(* Schneider Machine Expert - Basic project AWGC_ALGORITMA_COMMISSIONING, file version 3.0.0.0 *)
(* ProjectInformations: Name=New project *)

HARDWARE
  Cpu 0: TM221CE24R
  ModuleExtensionObject 0: TM3DI32K
  ModuleExtensionObject 1: TM3AI2H/G
  EthernetConfiguration: NetworkName=M221, IpAllocationMode=FixedAddress, IpAddress=0.0.0.0, SubnetMask=0.0.0.0
  SerialLineConfiguration: Baud=Baud19200, Parity=ParityEven, DataBits=DataBits8, StopBits=StopBits1, PhysicalMedium=PhysicalMediumRs485, TransmissionMode=TransmissionModeModbusRtu, SlaveId=1, Addressing=SlaveAddressing
  MastTask: UsePeriodScanMode=false, PeriodScan=100
  FastTask: Period=255
  CpuBehavior: StartingMode=StartAsPreviousState, AutoSaveRamOnEeprom=true, WatchdogPeriod=250

SYMBOLS  (address, symbol, comment, settings)
  %M0       SYSTEM_ENABLE  "Izin umum gerak"
  %M1       WATER_FAULT  "Fault sinyal level"
  %M2       FAULT_G1  "Fault pintu 1"
  %M3       FAULT_G2  "Fault pintu 2"
  %M4       FAULT_G3  "Fault pintu 3"
  %M5       SCADA_COMMISSIONING_OK  "Tombol SCADA commissioning OK"
  %M10      REVERSE_G1  "Arah encoder pintu 1 dibalik"
  %M11      REVERSE_G2  "Arah encoder pintu 2 dibalik"
  %M12      REVERSE_G3  "Arah encoder pintu 3 dibalik"
  %M100     G1_BIN_B0  "Binary bit 0 hasil Gray pintu 1"
  %M101     G1_BIN_B1  "Binary bit 1 hasil Gray pintu 1"
  %M102     G1_BIN_B2  "Binary bit 2 hasil Gray pintu 1"
  %M103     G1_BIN_B3  "Binary bit 3 hasil Gray pintu 1"
  %M104     G1_BIN_B4  "Binary bit 4 hasil Gray pintu 1"
  %M105     G1_BIN_B5  "Binary bit 5 hasil Gray pintu 1"
  %M106     G1_BIN_B6  "Binary bit 6 hasil Gray pintu 1"
  %M107     G1_BIN_B7  "Binary bit 7 hasil Gray pintu 1"
  %M110     G2_BIN_B0  "Binary bit 0 hasil Gray pintu 2"
  %M111     G2_BIN_B1  "Binary bit 1 hasil Gray pintu 2"
  %M112     G2_BIN_B2  "Binary bit 2 hasil Gray pintu 2"
  %M113     G2_BIN_B3  "Binary bit 3 hasil Gray pintu 2"
  %M114     G2_BIN_B4  "Binary bit 4 hasil Gray pintu 2"
  %M115     G2_BIN_B5  "Binary bit 5 hasil Gray pintu 2"
  %M116     G2_BIN_B6  "Binary bit 6 hasil Gray pintu 2"
  %M117     G2_BIN_B7  "Binary bit 7 hasil Gray pintu 2"
  %M120     G3_BIN_B0  "Binary bit 0 hasil Gray pintu 3"
  %M121     G3_BIN_B1  "Binary bit 1 hasil Gray pintu 3"
  %M122     G3_BIN_B2  "Binary bit 2 hasil Gray pintu 3"
  %M123     G3_BIN_B3  "Binary bit 3 hasil Gray pintu 3"
  %M124     G3_BIN_B4  "Binary bit 4 hasil Gray pintu 3"
  %M125     G3_BIN_B5  "Binary bit 5 hasil Gray pintu 3"
  %M126     G3_BIN_B6  "Binary bit 6 hasil Gray pintu 3"
  %M127     G3_BIN_B7  "Binary bit 7 hasil Gray pintu 3"
  %M200     AUTO_OPEN_REQ_G1  "Request auto buka G1"
  %M201     AUTO_CLOSE_REQ_G1  "Request auto tutup G1"
  %M202     AUTO_OPEN_REQ_G2  "Request auto buka G2"
  %M203     AUTO_CLOSE_REQ_G2  "Request auto tutup G2"
  %M204     AUTO_OPEN_REQ_G3  "Request auto buka G3"
  %M205     AUTO_CLOSE_REQ_G3  "Request auto tutup G3"
  %M210     MAN_OPEN_REQ_G1  "Request manual buka G1"
  %M211     MAN_CLOSE_REQ_G1  "Request manual tutup G1"
  %M212     MAN_OPEN_REQ_G2  "Request manual buka G2"
  %M213     MAN_CLOSE_REQ_G2  "Request manual tutup G2"
  %M214     MAN_OPEN_REQ_G3  "Request manual buka G3"
  %M215     MAN_CLOSE_REQ_G3  "Request manual tutup G3"
  %M6       SCADA_STOP  "BOOL RW: 1=STOP, 0=release stop; reset to STOP on first RUN"
  %M300     SCADA_SAFETY_OK  "Virtual input Safety OK dari SCADA"
  %M301     SCADA_LS_CLOSE_G1  "Virtual limit close gate 1"
  %M302     SCADA_LS_OPEN_G1  "Virtual limit open gate 1"
  %M303     SCADA_LS_CLOSE_G2  "Virtual limit close gate 2"
  %M304     SCADA_LS_OPEN_G2  "Virtual limit open gate 2"
  %M305     SCADA_LS_CLOSE_G3  "Virtual limit close gate 3"
  %M306     SCADA_LS_OPEN_G3  "Virtual limit open gate 3"
  %M307     SCADA_OL_G1_OK  "Virtual overload gate 1 OK"
  %M308     SCADA_OL_G2_OK  "Virtual overload gate 2 OK"
  %M309     SCADA_OL_G3_OK  "Virtual overload gate 3 OK"
  %M310     SIM_I0_10  "SIM ONLY virtual physical input I0.10"
  %M311     SIM_I0_11  "SIM ONLY virtual physical input I0.11"
  %M312     SIM_I0_12  "SIM ONLY virtual physical input I0.12"
  %M313     SIM_I0_13  "SIM ONLY virtual physical input I0.13"
  %M344     SCADA_MODE_AUTO  "Virtual mode AUTO dari SCADA"
  %M345     SIM_I1_25  "SIM ONLY virtual physical input I1.25"
  %M346     SIM_I1_26  "SIM ONLY virtual physical input I1.26"
  %M347     SIM_I1_27  "SIM ONLY virtual physical input I1.27"
  %M348     SIM_I1_28  "SIM ONLY virtual physical input I1.28"
  %M349     SIM_I1_29  "SIM ONLY virtual physical input I1.29"
  %M350     SIM_I1_30  "SIM ONLY virtual physical input I1.30"
  %M351     SCADA_RESET_FAULT  "Virtual reset fault dari SCADA"
  %M360     SIM_Q0_0  "SIM ONLY output mirror Q0.0; actual output always OFF"
  %M361     SIM_Q0_1  "SIM ONLY output mirror Q0.1; actual output always OFF"
  %M362     SIM_Q0_2  "SIM ONLY output mirror Q0.2; actual output always OFF"
  %M363     SIM_Q0_3  "SIM ONLY output mirror Q0.3; actual output always OFF"
  %M364     SIM_Q0_4  "SIM ONLY output mirror Q0.4; actual output always OFF"
  %M365     SIM_Q0_5  "SIM ONLY output mirror Q0.5; actual output always OFF"
  %M320     SIM_I1_0  "SIM ONLY virtual physical input I1.0"
  %M321     SIM_I1_1  "SIM ONLY virtual physical input I1.1"
  %M322     SIM_I1_2  "SIM ONLY virtual physical input I1.2"
  %M323     SIM_I1_3  "SIM ONLY virtual physical input I1.3"
  %M324     SIM_I1_4  "SIM ONLY virtual physical input I1.4"
  %M325     SIM_I1_5  "SIM ONLY virtual physical input I1.5"
  %M326     SIM_I1_6  "SIM ONLY virtual physical input I1.6"
  %M327     SIM_I1_7  "SIM ONLY virtual physical input I1.7"
  %M328     SIM_I1_8  "SIM ONLY virtual physical input I1.8"
  %M329     SIM_I1_9  "SIM ONLY virtual physical input I1.9"
  %M330     SIM_I1_10  "SIM ONLY virtual physical input I1.10"
  %M331     SIM_I1_11  "SIM ONLY virtual physical input I1.11"
  %M332     SIM_I1_12  "SIM ONLY virtual physical input I1.12"
  %M333     SIM_I1_13  "SIM ONLY virtual physical input I1.13"
  %M334     SIM_I1_14  "SIM ONLY virtual physical input I1.14"
  %M335     SIM_I1_15  "SIM ONLY virtual physical input I1.15"
  %M336     SIM_I1_16  "SIM ONLY virtual physical input I1.16"
  %M337     SIM_I1_17  "SIM ONLY virtual physical input I1.17"
  %M338     SIM_I1_18  "SIM ONLY virtual physical input I1.18"
  %M339     SIM_I1_19  "SIM ONLY virtual physical input I1.19"
  %M340     SIM_I1_20  "SIM ONLY virtual physical input I1.20"
  %M341     SIM_I1_21  "SIM ONLY virtual physical input I1.21"
  %M342     SIM_I1_22  "SIM ONLY virtual physical input I1.22"
  %M343     SIM_I1_23  "SIM ONLY virtual physical input I1.23"
  %M366     SIM_Q0_6  "SIM ONLY output mirror Q0.6; actual output always OFF"
  %M367     SIM_Q0_7  "SIM ONLY output mirror Q0.7; actual output always OFF"
  %M368     SIM_Q0_8  "SIM ONLY output mirror Q0.8; actual output always OFF"
  %M369     SIM_Q0_9  "SIM ONLY output mirror Q0.9; actual output always OFF"
  %M370     SCADA_ENABLE_SIM  "Virtual enable simulator dari SCADA"
  %S13      SB_FIRSTRUN  "Indicates the first controller cycle in RUN mode"
  %MW1      WATER_RANGE_MM  "Range sensor level mm"
  %MW2      LEVEL_RAW_COPY  "Salinan raw input level"
  %MW10     MAX_HEIGHT_G1_MM  "Tinggi maksimum pintu 1 mm"
  %MW11     MAX_HEIGHT_G2_MM  "Tinggi maksimum pintu 2 mm"
  %MW12     MAX_HEIGHT_G3_MM  "Tinggi maksimum pintu 3 mm"
  %MW13     DEADBAND_PCT  "Deadband posisi persen"
  %MW20     ENC_ZERO_G1  "Nilai encoder pintu 1 saat tertutup"
  %MW21     ENC_ZERO_G2  "Nilai encoder pintu 2 saat tertutup"
  %MW22     ENC_ZERO_G3  "Nilai encoder pintu 3 saat tertutup"
  %MW23     ENC_SPAN_G1  "Span count tertutup-terbuka G1"
  %MW24     ENC_SPAN_G2  "Span count tertutup-terbuka G2"
  %MW25     ENC_SPAN_G3  "Span count tertutup-terbuka G3"
  %MW30     ENC_BINARY_G1  "Nilai biner encoder G1"
  %MW31     ENC_BINARY_G2  "Nilai biner encoder G2"
  %MW32     ENC_BINARY_G3  "Nilai biner encoder G3"
  %MW33     POS_COUNT_G1  "Count posisi terkoreksi G1"
  %MW34     POS_COUNT_G2  "Count posisi terkoreksi G2"
  %MW35     POS_COUNT_G3  "Count posisi terkoreksi G3"
  %MW50     TARGET_PCT_G1  "Target bukaan G1 0-100 persen"
  %MW51     TARGET_PCT_G2  "Target bukaan G2 0-100 persen"
  %MW52     TARGET_PCT_G3  "Target bukaan G3 0-100 persen"
  %MW110    SIM_PROFILE_ID  "221 identifies simulation-only project"
  %MW111    SIM_PROFILE_VERSION  "4001 identifies simulation input mapping"
  %MF60     POSITION_G1_PCT  "Posisi G1 persen"
  %MF62     POSITION_G2_PCT  "Posisi G2 persen"
  %MF64     POSITION_G3_PCT  "Posisi G3 persen"
  %MF66     POSITION_G1_MM  "Posisi G1 mm"
  %MF68     POSITION_G2_MM  "Posisi G2 mm"
  %MF70     POSITION_G3_MM  "Posisi G3 mm"
  %MF72     WATER_LEVEL_MM  "Level air mm"
  %MF74     WATER_LEVEL_PCT  "Level air persen"
  %MF76     WATER_RANGE_REAL  "Range level dalam REAL"
  %MF80     TARGET_G1_REAL  "Target G1 dalam REAL"
  %MF82     TARGET_G2_REAL  "Target G2 dalam REAL"
  %MF84     TARGET_G3_REAL  "Target G3 dalam REAL"
  %MF86     DEADBAND_REAL  "Deadband dalam REAL"
  %MF88     OPEN_THRESHOLD_G1  "Ambang buka G1"
  %MF90     CLOSE_THRESHOLD_G1  "Ambang tutup G1"
  %MF92     OPEN_THRESHOLD_G2  "Ambang buka G2"
  %MF94     CLOSE_THRESHOLD_G2  "Ambang tutup G2"
  %MF96     OPEN_THRESHOLD_G3  "Ambang buka G3"
  %MF98     CLOSE_THRESHOLD_G3  "Ambang tutup G3"
  %I0.0     SAFETY_OK_IN  "Feedback rangkaian safety hardwired sehat"
  %I0.1     LS_CLOSE_G1  "Limit tertutup pintu 1"
  %I0.2     LS_OPEN_G1  "Limit terbuka pintu 1"
  %I0.3     LS_CLOSE_G2  "Limit tertutup pintu 2"
  %I0.4     LS_OPEN_G2  "Limit terbuka pintu 2"
  %I0.5     LS_CLOSE_G3  "Limit tertutup pintu 3"
  %I0.6     LS_OPEN_G3  "Limit terbuka pintu 3"
  %I0.7     OL_OK_G1  "Overload motor pintu 1 sehat"
  %I0.8     OL_OK_G2  "Overload motor pintu 2 sehat"
  %I0.9     OL_OK_G3  "Overload motor pintu 3 sehat"
  %I0.10    SPARE_I010  "Cadangan input"
  %I0.11    SPARE_I011  "Cadangan input"
  %I0.12    SPARE_I012  "Cadangan input"
  %I0.13    SPARE_I013  "Cadangan input"
  %Q0.0     OPEN_G1  "Relay kontaktor OPEN pintu 1"
  %Q0.1     CLOSE_G1  "Relay kontaktor CLOSE pintu 1"
  %Q0.2     OPEN_G2  "Relay kontaktor OPEN pintu 2"
  %Q0.3     CLOSE_G2  "Relay kontaktor CLOSE pintu 2"
  %Q0.4     OPEN_G3  "Relay kontaktor OPEN pintu 3"
  %Q0.5     CLOSE_G3  "Relay kontaktor CLOSE pintu 3"
  %I1.0     ENC_G1_GRAY_B0  "E6CP pintu 1 Gray bit 0"
  %I1.1     ENC_G1_GRAY_B1  "E6CP pintu 1 Gray bit 1"
  %I1.2     ENC_G1_GRAY_B2  "E6CP pintu 1 Gray bit 2"
  %I1.3     ENC_G1_GRAY_B3  "E6CP pintu 1 Gray bit 3"
  %I1.4     ENC_G1_GRAY_B4  "E6CP pintu 1 Gray bit 4"
  %I1.5     ENC_G1_GRAY_B5  "E6CP pintu 1 Gray bit 5"
  %I1.6     ENC_G1_GRAY_B6  "E6CP pintu 1 Gray bit 6"
  %I1.7     ENC_G1_GRAY_B7  "E6CP pintu 1 Gray bit 7"
  %I1.8     ENC_G2_GRAY_B0  "E6CP pintu 2 Gray bit 0"
  %I1.9     ENC_G2_GRAY_B1  "E6CP pintu 2 Gray bit 1"
  %I1.10    ENC_G2_GRAY_B2  "E6CP pintu 2 Gray bit 2"
  %I1.11    ENC_G2_GRAY_B3  "E6CP pintu 2 Gray bit 3"
  %I1.12    ENC_G2_GRAY_B4  "E6CP pintu 2 Gray bit 4"
  %I1.13    ENC_G2_GRAY_B5  "E6CP pintu 2 Gray bit 5"
  %I1.14    ENC_G2_GRAY_B6  "E6CP pintu 2 Gray bit 6"
  %I1.15    ENC_G2_GRAY_B7  "E6CP pintu 2 Gray bit 7"
  %I1.16    ENC_G3_GRAY_B0  "E6CP pintu 3 Gray bit 0"
  %I1.17    ENC_G3_GRAY_B1  "E6CP pintu 3 Gray bit 1"
  %I1.18    ENC_G3_GRAY_B2  "E6CP pintu 3 Gray bit 2"
  %I1.19    ENC_G3_GRAY_B3  "E6CP pintu 3 Gray bit 3"
  %I1.20    ENC_G3_GRAY_B4  "E6CP pintu 3 Gray bit 4"
  %I1.21    ENC_G3_GRAY_B5  "E6CP pintu 3 Gray bit 5"
  %I1.22    ENC_G3_GRAY_B6  "E6CP pintu 3 Gray bit 6"
  %I1.23    ENC_G3_GRAY_B7  "E6CP pintu 3 Gray bit 7"
  %I1.24    MODE_AUTO  "Selector 1=AUTO 0=MANUAL"
  %I1.25    MAN_OPEN_G1  "PB manual buka pintu 1"
  %I1.26    MAN_CLOSE_G1  "PB manual tutup pintu 1"
  %I1.27    MAN_OPEN_G2  "PB manual buka pintu 2"
  %I1.28    MAN_CLOSE_G2  "PB manual tutup pintu 2"
  %I1.29    MAN_OPEN_G3  "PB manual buka pintu 3"
  %I1.30    MAN_CLOSE_G3  "PB manual tutup pintu 3"
  %I1.31    RESET_FAULT  "PB reset fault"
  %IW2.0    LEVEL_RAW  "Sensor level 4-20 mA raw 4000-20000"  [Type=Type_4_20mA, Scope=Scope_Customized, Minimum=4000, Maximum=20000]

POU AWGC_3_PINTU_IL
  (* SectionNumber=1 *)

// Rung 0: SIM_COLD_RESET_M369
// SIMULATOR ONLY. Physical outputs forced OFF. Do not use for plant operation.
  LD %S13                 (* SB_FIRSTRUN *)
  R %M369                 (* SIM_Q0_9 *)
  // as ST:
  //   IF SB_FIRSTRUN THEN SIM_Q0_9 := FALSE; END_IF;

// Rung 1: SIM_COLD_RESET_M368
// SIMULATOR ONLY. Physical outputs forced OFF. Do not use for plant operation.
  LD %S13                 (* SB_FIRSTRUN *)
  R %M368                 (* SIM_Q0_8 *)
  // as ST:
  //   IF SB_FIRSTRUN THEN SIM_Q0_8 := FALSE; END_IF;

// Rung 2: SIM_COLD_RESET_M367
// SIMULATOR ONLY. Physical outputs forced OFF. Do not use for plant operation.
  LD %S13                 (* SB_FIRSTRUN *)
  R %M367                 (* SIM_Q0_7 *)
  // as ST:
  //   IF SB_FIRSTRUN THEN SIM_Q0_7 := FALSE; END_IF;

// Rung 3: SIM_COLD_RESET_M366
// SIMULATOR ONLY. Physical outputs forced OFF. Do not use for plant operation.
  LD %S13                 (* SB_FIRSTRUN *)
  R %M366                 (* SIM_Q0_6 *)
  // as ST:
  //   IF SB_FIRSTRUN THEN SIM_Q0_6 := FALSE; END_IF;

// Rung 4: SIM_COLD_RESET_M365
// SIMULATOR ONLY. Physical outputs forced OFF. Do not use for plant operation.
  LD %S13                 (* SB_FIRSTRUN *)
  R %M365                 (* SIM_Q0_5 *)
  // as ST:
  //   IF SB_FIRSTRUN THEN SIM_Q0_5 := FALSE; END_IF;

// Rung 5: SIM_COLD_RESET_M364
// SIMULATOR ONLY. Physical outputs forced OFF. Do not use for plant operation.
  LD %S13                 (* SB_FIRSTRUN *)
  R %M364                 (* SIM_Q0_4 *)
  // as ST:
  //   IF SB_FIRSTRUN THEN SIM_Q0_4 := FALSE; END_IF;

// Rung 6: SIM_COLD_RESET_M363
// SIMULATOR ONLY. Physical outputs forced OFF. Do not use for plant operation.
  LD %S13                 (* SB_FIRSTRUN *)
  R %M363                 (* SIM_Q0_3 *)
  // as ST:
  //   IF SB_FIRSTRUN THEN SIM_Q0_3 := FALSE; END_IF;

// Rung 7: SIM_COLD_RESET_M362
// SIMULATOR ONLY. Physical outputs forced OFF. Do not use for plant operation.
  LD %S13                 (* SB_FIRSTRUN *)
  R %M362                 (* SIM_Q0_2 *)
  // as ST:
  //   IF SB_FIRSTRUN THEN SIM_Q0_2 := FALSE; END_IF;

// Rung 8: SIM_COLD_RESET_M361
// SIMULATOR ONLY. Physical outputs forced OFF. Do not use for plant operation.
  LD %S13                 (* SB_FIRSTRUN *)
  R %M361                 (* SIM_Q0_1 *)
  // as ST:
  //   IF SB_FIRSTRUN THEN SIM_Q0_1 := FALSE; END_IF;

// Rung 9: SIM_COLD_RESET_M360
// SIMULATOR ONLY. Physical outputs forced OFF. Do not use for plant operation.
  LD %S13                 (* SB_FIRSTRUN *)
  R %M360                 (* SIM_Q0_0 *)
  // as ST:
  //   IF SB_FIRSTRUN THEN SIM_Q0_0 := FALSE; END_IF;

// Rung 10: SIM_COLD_RESET_M351
// SIMULATOR ONLY. Physical outputs forced OFF. Do not use for plant operation.
  LD %S13                 (* SB_FIRSTRUN *)
  R %M351                 (* SCADA_RESET_FAULT *)
  // as ST:
  //   IF SB_FIRSTRUN THEN SCADA_RESET_FAULT := FALSE; END_IF;

// Rung 11: SIM_COLD_RESET_M350
// SIMULATOR ONLY. Physical outputs forced OFF. Do not use for plant operation.
  LD %S13                 (* SB_FIRSTRUN *)
  R %M350                 (* SIM_I1_30 *)
  // as ST:
  //   IF SB_FIRSTRUN THEN SIM_I1_30 := FALSE; END_IF;

// Rung 12: SIM_COLD_RESET_M349
// SIMULATOR ONLY. Physical outputs forced OFF. Do not use for plant operation.
  LD %S13                 (* SB_FIRSTRUN *)
  R %M349                 (* SIM_I1_29 *)
  // as ST:
  //   IF SB_FIRSTRUN THEN SIM_I1_29 := FALSE; END_IF;

// Rung 13: SIM_COLD_RESET_M348
// SIMULATOR ONLY. Physical outputs forced OFF. Do not use for plant operation.
  LD %S13                 (* SB_FIRSTRUN *)
  R %M348                 (* SIM_I1_28 *)
  // as ST:
  //   IF SB_FIRSTRUN THEN SIM_I1_28 := FALSE; END_IF;

// Rung 14: SIM_COLD_RESET_M347
// SIMULATOR ONLY. Physical outputs forced OFF. Do not use for plant operation.
  LD %S13                 (* SB_FIRSTRUN *)
  R %M347                 (* SIM_I1_27 *)
  // as ST:
  //   IF SB_FIRSTRUN THEN SIM_I1_27 := FALSE; END_IF;

// Rung 15: SIM_COLD_RESET_M346
// SIMULATOR ONLY. Physical outputs forced OFF. Do not use for plant operation.
  LD %S13                 (* SB_FIRSTRUN *)
  R %M346                 (* SIM_I1_26 *)
  // as ST:
  //   IF SB_FIRSTRUN THEN SIM_I1_26 := FALSE; END_IF;

// Rung 16: SIM_COLD_RESET_M345
// SIMULATOR ONLY. Physical outputs forced OFF. Do not use for plant operation.
  LD %S13                 (* SB_FIRSTRUN *)
  R %M345                 (* SIM_I1_25 *)
  // as ST:
  //   IF SB_FIRSTRUN THEN SIM_I1_25 := FALSE; END_IF;

// Rung 17: SIM_COLD_RESET_M344
// SIMULATOR ONLY. Physical outputs forced OFF. Do not use for plant operation.
  LD %S13                 (* SB_FIRSTRUN *)
  R %M344                 (* SCADA_MODE_AUTO *)
  // as ST:
  //   IF SB_FIRSTRUN THEN SCADA_MODE_AUTO := FALSE; END_IF;

// Rung 18: SIM_COLD_RESET_M343
// SIMULATOR ONLY. Physical outputs forced OFF. Do not use for plant operation.
  LD %S13                 (* SB_FIRSTRUN *)
  R %M343                 (* SIM_I1_23 *)
  // as ST:
  //   IF SB_FIRSTRUN THEN SIM_I1_23 := FALSE; END_IF;

// Rung 19: SIM_COLD_RESET_M342
// SIMULATOR ONLY. Physical outputs forced OFF. Do not use for plant operation.
  LD %S13                 (* SB_FIRSTRUN *)
  R %M342                 (* SIM_I1_22 *)
  // as ST:
  //   IF SB_FIRSTRUN THEN SIM_I1_22 := FALSE; END_IF;

// Rung 20: SIM_COLD_RESET_M341
// SIMULATOR ONLY. Physical outputs forced OFF. Do not use for plant operation.
  LD %S13                 (* SB_FIRSTRUN *)
  R %M341                 (* SIM_I1_21 *)
  // as ST:
  //   IF SB_FIRSTRUN THEN SIM_I1_21 := FALSE; END_IF;

// Rung 21: SIM_COLD_RESET_M340
// SIMULATOR ONLY. Physical outputs forced OFF. Do not use for plant operation.
  LD %S13                 (* SB_FIRSTRUN *)
  R %M340                 (* SIM_I1_20 *)
  // as ST:
  //   IF SB_FIRSTRUN THEN SIM_I1_20 := FALSE; END_IF;

// Rung 22: SIM_COLD_RESET_M339
// SIMULATOR ONLY. Physical outputs forced OFF. Do not use for plant operation.
  LD %S13                 (* SB_FIRSTRUN *)
  R %M339                 (* SIM_I1_19 *)
  // as ST:
  //   IF SB_FIRSTRUN THEN SIM_I1_19 := FALSE; END_IF;

// Rung 23: SIM_COLD_RESET_M338
// SIMULATOR ONLY. Physical outputs forced OFF. Do not use for plant operation.
  LD %S13                 (* SB_FIRSTRUN *)
  R %M338                 (* SIM_I1_18 *)
  // as ST:
  //   IF SB_FIRSTRUN THEN SIM_I1_18 := FALSE; END_IF;

// Rung 24: SIM_COLD_RESET_M337
// SIMULATOR ONLY. Physical outputs forced OFF. Do not use for plant operation.
  LD %S13                 (* SB_FIRSTRUN *)
  R %M337                 (* SIM_I1_17 *)
  // as ST:
  //   IF SB_FIRSTRUN THEN SIM_I1_17 := FALSE; END_IF;

// Rung 25: SIM_COLD_RESET_M336
// SIMULATOR ONLY. Physical outputs forced OFF. Do not use for plant operation.
  LD %S13                 (* SB_FIRSTRUN *)
  R %M336                 (* SIM_I1_16 *)
  // as ST:
  //   IF SB_FIRSTRUN THEN SIM_I1_16 := FALSE; END_IF;

// Rung 26: SIM_COLD_RESET_M335
// SIMULATOR ONLY. Physical outputs forced OFF. Do not use for plant operation.
  LD %S13                 (* SB_FIRSTRUN *)
  R %M335                 (* SIM_I1_15 *)
  // as ST:
  //   IF SB_FIRSTRUN THEN SIM_I1_15 := FALSE; END_IF;

// Rung 27: SIM_COLD_RESET_M334
// SIMULATOR ONLY. Physical outputs forced OFF. Do not use for plant operation.
  LD %S13                 (* SB_FIRSTRUN *)
  R %M334                 (* SIM_I1_14 *)
  // as ST:
  //   IF SB_FIRSTRUN THEN SIM_I1_14 := FALSE; END_IF;

// Rung 28: SIM_COLD_RESET_M333
// SIMULATOR ONLY. Physical outputs forced OFF. Do not use for plant operation.
  LD %S13                 (* SB_FIRSTRUN *)
  R %M333                 (* SIM_I1_13 *)
  // as ST:
  //   IF SB_FIRSTRUN THEN SIM_I1_13 := FALSE; END_IF;

// Rung 29: SIM_COLD_RESET_M332
// SIMULATOR ONLY. Physical outputs forced OFF. Do not use for plant operation.
  LD %S13                 (* SB_FIRSTRUN *)
  R %M332                 (* SIM_I1_12 *)
  // as ST:
  //   IF SB_FIRSTRUN THEN SIM_I1_12 := FALSE; END_IF;

// Rung 30: SIM_COLD_RESET_M331
// SIMULATOR ONLY. Physical outputs forced OFF. Do not use for plant operation.
  LD %S13                 (* SB_FIRSTRUN *)
  R %M331                 (* SIM_I1_11 *)
  // as ST:
  //   IF SB_FIRSTRUN THEN SIM_I1_11 := FALSE; END_IF;

// Rung 31: SIM_COLD_RESET_M330
// SIMULATOR ONLY. Physical outputs forced OFF. Do not use for plant operation.
  LD %S13                 (* SB_FIRSTRUN *)
  R %M330                 (* SIM_I1_10 *)
  // as ST:
  //   IF SB_FIRSTRUN THEN SIM_I1_10 := FALSE; END_IF;

// Rung 32: SIM_COLD_RESET_M329
// SIMULATOR ONLY. Physical outputs forced OFF. Do not use for plant operation.
  LD %S13                 (* SB_FIRSTRUN *)
  R %M329                 (* SIM_I1_9 *)
  // as ST:
  //   IF SB_FIRSTRUN THEN SIM_I1_9 := FALSE; END_IF;

// Rung 33: SIM_COLD_RESET_M328
// SIMULATOR ONLY. Physical outputs forced OFF. Do not use for plant operation.
  LD %S13                 (* SB_FIRSTRUN *)
  R %M328                 (* SIM_I1_8 *)
  // as ST:
  //   IF SB_FIRSTRUN THEN SIM_I1_8 := FALSE; END_IF;

// Rung 34: SIM_COLD_RESET_M327
// SIMULATOR ONLY. Physical outputs forced OFF. Do not use for plant operation.
  LD %S13                 (* SB_FIRSTRUN *)
  R %M327                 (* SIM_I1_7 *)
  // as ST:
  //   IF SB_FIRSTRUN THEN SIM_I1_7 := FALSE; END_IF;

// Rung 35: SIM_COLD_RESET_M326
// SIMULATOR ONLY. Physical outputs forced OFF. Do not use for plant operation.
  LD %S13                 (* SB_FIRSTRUN *)
  R %M326                 (* SIM_I1_6 *)
  // as ST:
  //   IF SB_FIRSTRUN THEN SIM_I1_6 := FALSE; END_IF;

// Rung 36: SIM_COLD_RESET_M325
// SIMULATOR ONLY. Physical outputs forced OFF. Do not use for plant operation.
  LD %S13                 (* SB_FIRSTRUN *)
  R %M325                 (* SIM_I1_5 *)
  // as ST:
  //   IF SB_FIRSTRUN THEN SIM_I1_5 := FALSE; END_IF;

// Rung 37: SIM_COLD_RESET_M324
// SIMULATOR ONLY. Physical outputs forced OFF. Do not use for plant operation.
  LD %S13                 (* SB_FIRSTRUN *)
  R %M324                 (* SIM_I1_4 *)
  // as ST:
  //   IF SB_FIRSTRUN THEN SIM_I1_4 := FALSE; END_IF;

// Rung 38: SIM_COLD_RESET_M323
// SIMULATOR ONLY. Physical outputs forced OFF. Do not use for plant operation.
  LD %S13                 (* SB_FIRSTRUN *)
  R %M323                 (* SIM_I1_3 *)
  // as ST:
  //   IF SB_FIRSTRUN THEN SIM_I1_3 := FALSE; END_IF;

// Rung 39: SIM_COLD_RESET_M322
// SIMULATOR ONLY. Physical outputs forced OFF. Do not use for plant operation.
  LD %S13                 (* SB_FIRSTRUN *)
  R %M322                 (* SIM_I1_2 *)
  // as ST:
  //   IF SB_FIRSTRUN THEN SIM_I1_2 := FALSE; END_IF;

// Rung 40: SIM_COLD_RESET_M321
// SIMULATOR ONLY. Physical outputs forced OFF. Do not use for plant operation.
  LD %S13                 (* SB_FIRSTRUN *)
  R %M321                 (* SIM_I1_1 *)
  // as ST:
  //   IF SB_FIRSTRUN THEN SIM_I1_1 := FALSE; END_IF;

// Rung 41: SIM_COLD_RESET_M320
// SIMULATOR ONLY. Physical outputs forced OFF. Do not use for plant operation.
  LD %S13                 (* SB_FIRSTRUN *)
  R %M320                 (* SIM_I1_0 *)
  // as ST:
  //   IF SB_FIRSTRUN THEN SIM_I1_0 := FALSE; END_IF;

// Rung 42: SIM_COLD_RESET_M313
// SIMULATOR ONLY. Physical outputs forced OFF. Do not use for plant operation.
  LD %S13                 (* SB_FIRSTRUN *)
  R %M313                 (* SIM_I0_13 *)
  // as ST:
  //   IF SB_FIRSTRUN THEN SIM_I0_13 := FALSE; END_IF;

// Rung 43: SIM_COLD_RESET_M312
// SIMULATOR ONLY. Physical outputs forced OFF. Do not use for plant operation.
  LD %S13                 (* SB_FIRSTRUN *)
  R %M312                 (* SIM_I0_12 *)
  // as ST:
  //   IF SB_FIRSTRUN THEN SIM_I0_12 := FALSE; END_IF;

// Rung 44: SIM_COLD_RESET_M311
// SIMULATOR ONLY. Physical outputs forced OFF. Do not use for plant operation.
  LD %S13                 (* SB_FIRSTRUN *)
  R %M311                 (* SIM_I0_11 *)
  // as ST:
  //   IF SB_FIRSTRUN THEN SIM_I0_11 := FALSE; END_IF;

// Rung 45: SIM_COLD_RESET_M310
// SIMULATOR ONLY. Physical outputs forced OFF. Do not use for plant operation.
  LD %S13                 (* SB_FIRSTRUN *)
  R %M310                 (* SIM_I0_10 *)
  // as ST:
  //   IF SB_FIRSTRUN THEN SIM_I0_10 := FALSE; END_IF;

// Rung 46: SIM_COLD_RESET_M309
// SIMULATOR ONLY. Physical outputs forced OFF. Do not use for plant operation.
  LD %S13                 (* SB_FIRSTRUN *)
  R %M309                 (* SCADA_OL_G3_OK *)
  // as ST:
  //   IF SB_FIRSTRUN THEN SCADA_OL_G3_OK := FALSE; END_IF;

// Rung 47: SIM_COLD_RESET_M308
// SIMULATOR ONLY. Physical outputs forced OFF. Do not use for plant operation.
  LD %S13                 (* SB_FIRSTRUN *)
  R %M308                 (* SCADA_OL_G2_OK *)
  // as ST:
  //   IF SB_FIRSTRUN THEN SCADA_OL_G2_OK := FALSE; END_IF;

// Rung 48: SIM_COLD_RESET_M307
// SIMULATOR ONLY. Physical outputs forced OFF. Do not use for plant operation.
  LD %S13                 (* SB_FIRSTRUN *)
  R %M307                 (* SCADA_OL_G1_OK *)
  // as ST:
  //   IF SB_FIRSTRUN THEN SCADA_OL_G1_OK := FALSE; END_IF;

// Rung 49: SIM_COLD_RESET_M306
// SIMULATOR ONLY. Physical outputs forced OFF. Do not use for plant operation.
  LD %S13                 (* SB_FIRSTRUN *)
  R %M306                 (* SCADA_LS_OPEN_G3 *)
  // as ST:
  //   IF SB_FIRSTRUN THEN SCADA_LS_OPEN_G3 := FALSE; END_IF;

// Rung 50: SIM_COLD_RESET_M305
// SIMULATOR ONLY. Physical outputs forced OFF. Do not use for plant operation.
  LD %S13                 (* SB_FIRSTRUN *)
  R %M305                 (* SCADA_LS_CLOSE_G3 *)
  // as ST:
  //   IF SB_FIRSTRUN THEN SCADA_LS_CLOSE_G3 := FALSE; END_IF;

// Rung 51: SIM_COLD_RESET_M304
// SIMULATOR ONLY. Physical outputs forced OFF. Do not use for plant operation.
  LD %S13                 (* SB_FIRSTRUN *)
  R %M304                 (* SCADA_LS_OPEN_G2 *)
  // as ST:
  //   IF SB_FIRSTRUN THEN SCADA_LS_OPEN_G2 := FALSE; END_IF;

// Rung 52: SIM_COLD_RESET_M303
// SIMULATOR ONLY. Physical outputs forced OFF. Do not use for plant operation.
  LD %S13                 (* SB_FIRSTRUN *)
  R %M303                 (* SCADA_LS_CLOSE_G2 *)
  // as ST:
  //   IF SB_FIRSTRUN THEN SCADA_LS_CLOSE_G2 := FALSE; END_IF;

// Rung 53: SIM_COLD_RESET_M302
// SIMULATOR ONLY. Physical outputs forced OFF. Do not use for plant operation.
  LD %S13                 (* SB_FIRSTRUN *)
  R %M302                 (* SCADA_LS_OPEN_G1 *)
  // as ST:
  //   IF SB_FIRSTRUN THEN SCADA_LS_OPEN_G1 := FALSE; END_IF;

// Rung 54: SIM_COLD_RESET_M301
// SIMULATOR ONLY. Physical outputs forced OFF. Do not use for plant operation.
  LD %S13                 (* SB_FIRSTRUN *)
  R %M301                 (* SCADA_LS_CLOSE_G1 *)
  // as ST:
  //   IF SB_FIRSTRUN THEN SCADA_LS_CLOSE_G1 := FALSE; END_IF;

// Rung 55: SIM_COLD_RESET_M300
// SIMULATOR ONLY. Physical outputs forced OFF. Do not use for plant operation.
  LD %S13                 (* SB_FIRSTRUN *)
  R %M300                 (* SCADA_SAFETY_OK *)
  // as ST:
  //   IF SB_FIRSTRUN THEN SCADA_SAFETY_OK := FALSE; END_IF;

// Rung 56: SIM_COLD_RESET_M370
// SIMULATOR ONLY. Physical outputs forced OFF. Do not use for plant operation.
  LD %S13                 (* SB_FIRSTRUN *)
  R %M370                 (* SCADA_ENABLE_SIM *)
  // as ST:
  //   IF SB_FIRSTRUN THEN SCADA_ENABLE_SIM := FALSE; END_IF;

// Rung 57: SIM_COLD_RESET_M5
// SIMULATOR ONLY. Physical outputs forced OFF. Do not use for plant operation.
  LD %S13                 (* SB_FIRSTRUN *)
  R %M5                   (* SCADA_COMMISSIONING_OK *)
  // as ST:
  //   IF SB_FIRSTRUN THEN SCADA_COMMISSIONING_OK := FALSE; END_IF;

// Rung 58: SIM_PROFILE_ID
// SIMULATOR ONLY. Physical outputs forced OFF. Do not use for plant operation.
  LD 1
  [ %MW110 := 221 ]       (* SIM_PROFILE_ID *)
  // as ST:
  //   SIM_PROFILE_ID := 221;

// Rung 59: SIM_PROFILE_VERSION
// SIMULATOR ONLY. Physical outputs forced OFF. Do not use for plant operation.
  LD 1
  [ %MW111 := 4001 ]      (* SIM_PROFILE_VERSION *)
  // as ST:
  //   SIM_PROFILE_VERSION := 4001;

// Rung 60: REV3_SCADA_VERSION
// REV3 SCADA compatibility marker; not authentication.
  LD 1
  [ %MW111 := 3001 ]      (* SIM_PROFILE_VERSION *)
  // as ST:
  //   SIM_PROFILE_VERSION := 3001;

// Rung 61: REV3_SCADA_ID
// REV3 SCADA compatibility marker; not authentication.
  LD 1
  [ %MW110 := 221 ]       (* SIM_PROFILE_ID *)
  // as ST:
  //   SIM_PROFILE_ID := 221;

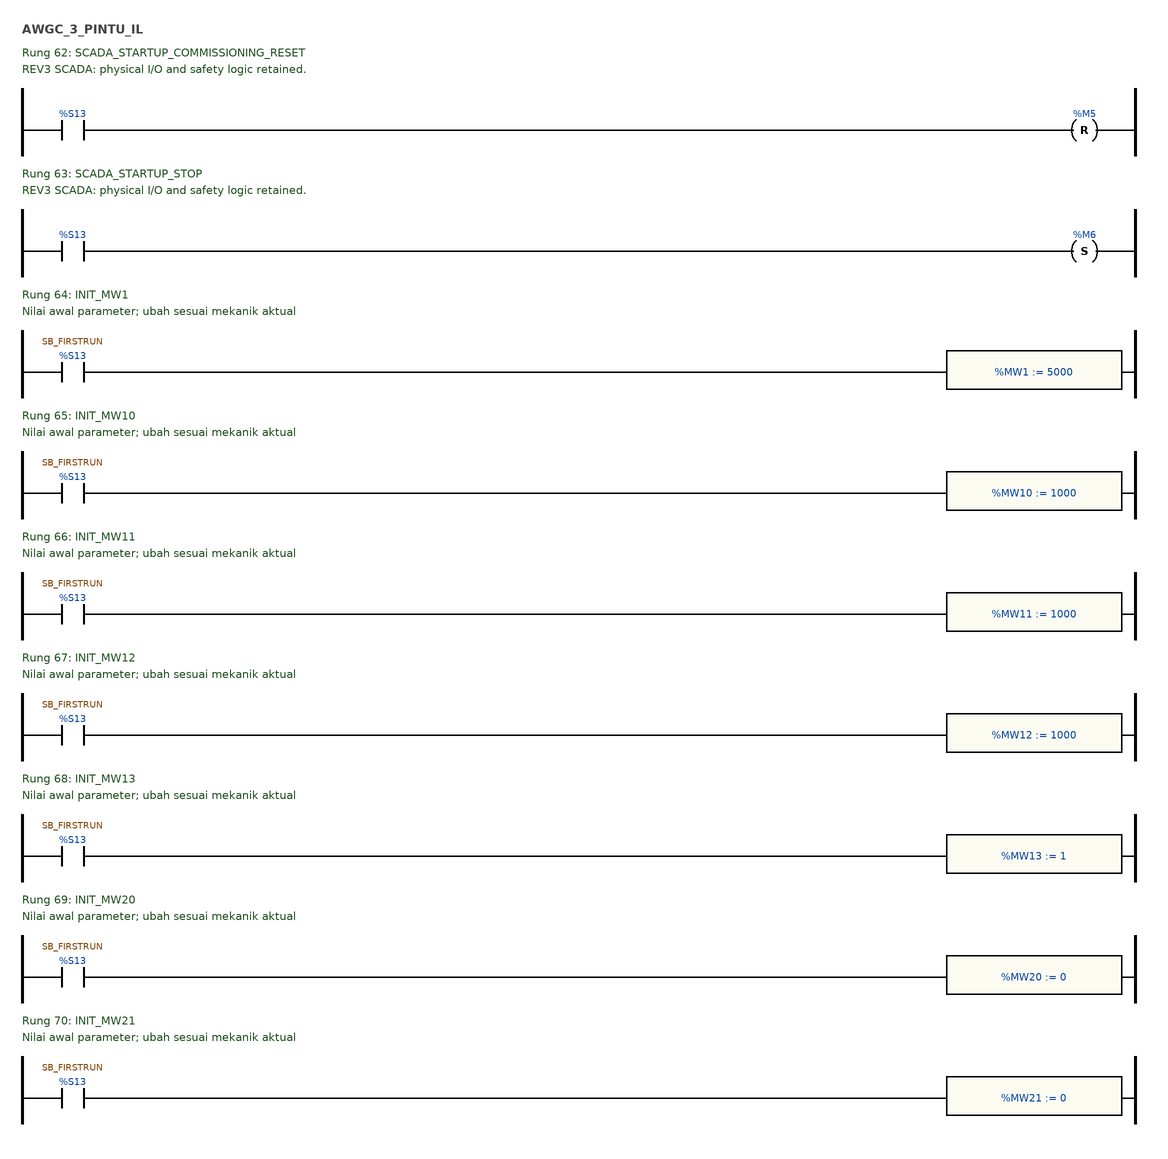

// Rung 62: SCADA_STARTUP_COMMISSIONING_RESET
// REV3 SCADA: physical I/O and safety logic retained.
  LD %S13                 (* SB_FIRSTRUN *)
  R %M5                   (* SCADA_COMMISSIONING_OK *)
  // as ST:
  //   IF SB_FIRSTRUN THEN SCADA_COMMISSIONING_OK := FALSE; END_IF;

// Rung 63: SCADA_STARTUP_STOP
// REV3 SCADA: physical I/O and safety logic retained.
  LD %S13                 (* SB_FIRSTRUN *)
  S %M6                   (* SCADA_STOP *)
  // as ST:
  //   IF SB_FIRSTRUN THEN SCADA_STOP := TRUE; END_IF;

// Rung 64: INIT_MW1
// Nilai awal parameter; ubah sesuai mekanik aktual
  LD %S13                 (* SB_FIRSTRUN *)
  [ %MW1 := 5000 ]        (* WATER_RANGE_MM *)
  // as ST:
  //   IF SB_FIRSTRUN THEN WATER_RANGE_MM := 5000; END_IF;

// Rung 65: INIT_MW10
// Nilai awal parameter; ubah sesuai mekanik aktual
  LD %S13                 (* SB_FIRSTRUN *)
  [ %MW10 := 1000 ]       (* MAX_HEIGHT_G1_MM *)
  // as ST:
  //   IF SB_FIRSTRUN THEN MAX_HEIGHT_G1_MM := 1000; END_IF;

// Rung 66: INIT_MW11
// Nilai awal parameter; ubah sesuai mekanik aktual
  LD %S13                 (* SB_FIRSTRUN *)
  [ %MW11 := 1000 ]       (* MAX_HEIGHT_G2_MM *)
  // as ST:
  //   IF SB_FIRSTRUN THEN MAX_HEIGHT_G2_MM := 1000; END_IF;

// Rung 67: INIT_MW12
// Nilai awal parameter; ubah sesuai mekanik aktual
  LD %S13                 (* SB_FIRSTRUN *)
  [ %MW12 := 1000 ]       (* MAX_HEIGHT_G3_MM *)
  // as ST:
  //   IF SB_FIRSTRUN THEN MAX_HEIGHT_G3_MM := 1000; END_IF;

// Rung 68: INIT_MW13
// Nilai awal parameter; ubah sesuai mekanik aktual
  LD %S13                 (* SB_FIRSTRUN *)
  [ %MW13 := 1 ]          (* DEADBAND_PCT *)
  // as ST:
  //   IF SB_FIRSTRUN THEN DEADBAND_PCT := 1; END_IF;

// Rung 69: INIT_MW20
// Nilai awal parameter; ubah sesuai mekanik aktual
  LD %S13                 (* SB_FIRSTRUN *)
  [ %MW20 := 0 ]          (* ENC_ZERO_G1 *)
  // as ST:
  //   IF SB_FIRSTRUN THEN ENC_ZERO_G1 := 0; END_IF;

// Rung 70: INIT_MW21
// Nilai awal parameter; ubah sesuai mekanik aktual
  LD %S13                 (* SB_FIRSTRUN *)
  [ %MW21 := 0 ]          (* ENC_ZERO_G2 *)
  // as ST:
  //   IF SB_FIRSTRUN THEN ENC_ZERO_G2 := 0; END_IF;

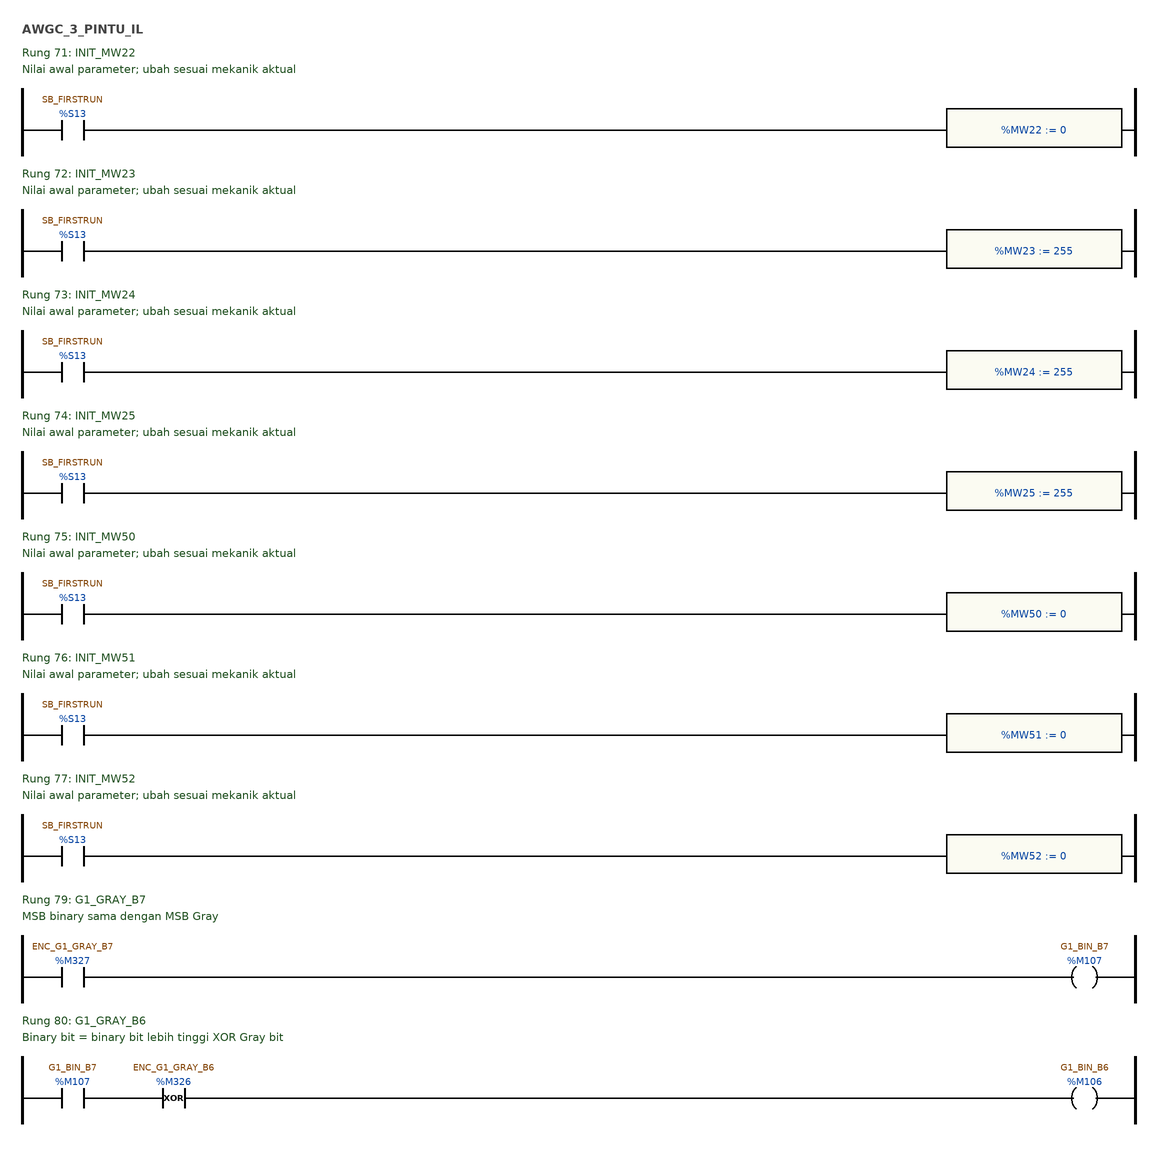

// Rung 71: INIT_MW22
// Nilai awal parameter; ubah sesuai mekanik aktual
  LD %S13                 (* SB_FIRSTRUN *)
  [ %MW22 := 0 ]          (* ENC_ZERO_G3 *)
  // as ST:
  //   IF SB_FIRSTRUN THEN ENC_ZERO_G3 := 0; END_IF;

// Rung 72: INIT_MW23
// Nilai awal parameter; ubah sesuai mekanik aktual
  LD %S13                 (* SB_FIRSTRUN *)
  [ %MW23 := 255 ]        (* ENC_SPAN_G1 *)
  // as ST:
  //   IF SB_FIRSTRUN THEN ENC_SPAN_G1 := 255; END_IF;

// Rung 73: INIT_MW24
// Nilai awal parameter; ubah sesuai mekanik aktual
  LD %S13                 (* SB_FIRSTRUN *)
  [ %MW24 := 255 ]        (* ENC_SPAN_G2 *)
  // as ST:
  //   IF SB_FIRSTRUN THEN ENC_SPAN_G2 := 255; END_IF;

// Rung 74: INIT_MW25
// Nilai awal parameter; ubah sesuai mekanik aktual
  LD %S13                 (* SB_FIRSTRUN *)
  [ %MW25 := 255 ]        (* ENC_SPAN_G3 *)
  // as ST:
  //   IF SB_FIRSTRUN THEN ENC_SPAN_G3 := 255; END_IF;

// Rung 75: INIT_MW50
// Nilai awal parameter; ubah sesuai mekanik aktual
  LD %S13                 (* SB_FIRSTRUN *)
  [ %MW50 := 0 ]          (* TARGET_PCT_G1 *)
  // as ST:
  //   IF SB_FIRSTRUN THEN TARGET_PCT_G1 := 0; END_IF;

// Rung 76: INIT_MW51
// Nilai awal parameter; ubah sesuai mekanik aktual
  LD %S13                 (* SB_FIRSTRUN *)
  [ %MW51 := 0 ]          (* TARGET_PCT_G2 *)
  // as ST:
  //   IF SB_FIRSTRUN THEN TARGET_PCT_G2 := 0; END_IF;

// Rung 77: INIT_MW52
// Nilai awal parameter; ubah sesuai mekanik aktual
  LD %S13                 (* SB_FIRSTRUN *)
  [ %MW52 := 0 ]          (* TARGET_PCT_G3 *)
  // as ST:
  //   IF SB_FIRSTRUN THEN TARGET_PCT_G3 := 0; END_IF;

// Rung 78: SYSTEM_PERMISSIVE_SIM
// SIMULATOR ONLY. Physical outputs forced OFF. Do not use for plant operation.
  LD %M300                (* SCADA_SAFETY_OK *)
  AND %M307               (* SCADA_OL_G1_OK *)
  AND %M308               (* SCADA_OL_G2_OK *)
  AND %M309               (* SCADA_OL_G3_OK *)
  AND %M5                 (* SCADA_COMMISSIONING_OK *)
  AND %M370               (* SCADA_ENABLE_SIM *)
  ST %M0                  (* SYSTEM_ENABLE *)
  // as ST:
  //   SYSTEM_ENABLE := SCADA_SAFETY_OK AND SCADA_OL_G1_OK AND SCADA_OL_G2_OK AND SCADA_OL_G3_OK AND SCADA_COMMISSIONING_OK AND SCADA_ENABLE_SIM;

// Rung 79: G1_GRAY_B7
// MSB binary sama dengan MSB Gray
  LD %M327                (* SIM_I1_7 *)
  ST %M107                (* G1_BIN_B7 *)
  // as ST:
  //   G1_BIN_B7 := SIM_I1_7;

// Rung 80: G1_GRAY_B6
// Binary bit = binary bit lebih tinggi XOR Gray bit
  LD %M107                (* G1_BIN_B7 *)
  XOR %M326               (* SIM_I1_6 *)
  ST %M106                (* G1_BIN_B6 *)
  // as ST:
  //   G1_BIN_B6 := G1_BIN_B7 XOR SIM_I1_6;

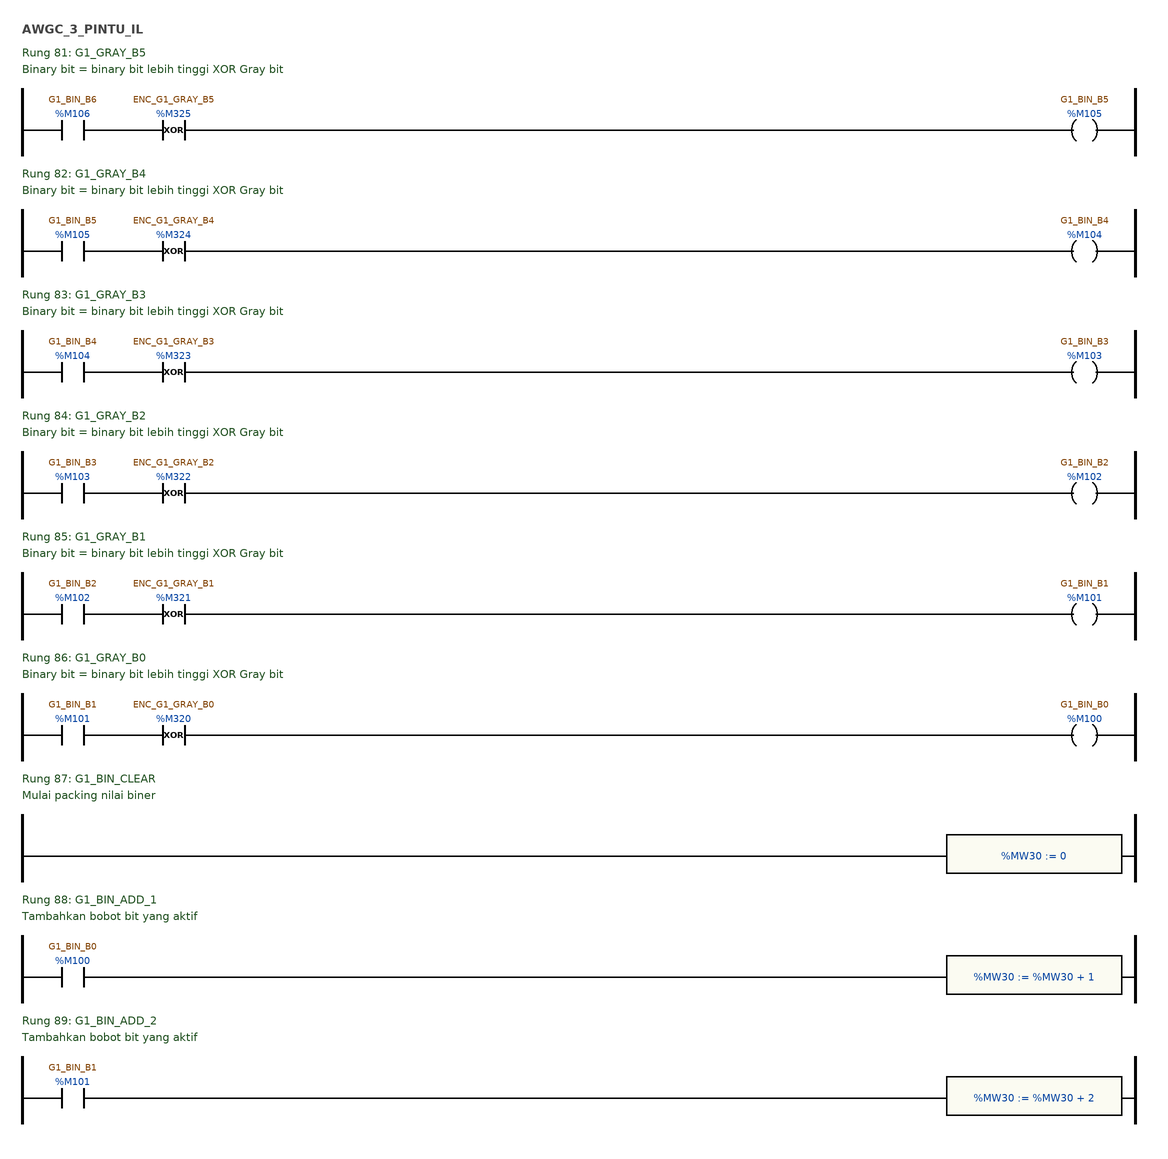

// Rung 81: G1_GRAY_B5
// Binary bit = binary bit lebih tinggi XOR Gray bit
  LD %M106                (* G1_BIN_B6 *)
  XOR %M325               (* SIM_I1_5 *)
  ST %M105                (* G1_BIN_B5 *)
  // as ST:
  //   G1_BIN_B5 := G1_BIN_B6 XOR SIM_I1_5;

// Rung 82: G1_GRAY_B4
// Binary bit = binary bit lebih tinggi XOR Gray bit
  LD %M105                (* G1_BIN_B5 *)
  XOR %M324               (* SIM_I1_4 *)
  ST %M104                (* G1_BIN_B4 *)
  // as ST:
  //   G1_BIN_B4 := G1_BIN_B5 XOR SIM_I1_4;

// Rung 83: G1_GRAY_B3
// Binary bit = binary bit lebih tinggi XOR Gray bit
  LD %M104                (* G1_BIN_B4 *)
  XOR %M323               (* SIM_I1_3 *)
  ST %M103                (* G1_BIN_B3 *)
  // as ST:
  //   G1_BIN_B3 := G1_BIN_B4 XOR SIM_I1_3;

// Rung 84: G1_GRAY_B2
// Binary bit = binary bit lebih tinggi XOR Gray bit
  LD %M103                (* G1_BIN_B3 *)
  XOR %M322               (* SIM_I1_2 *)
  ST %M102                (* G1_BIN_B2 *)
  // as ST:
  //   G1_BIN_B2 := G1_BIN_B3 XOR SIM_I1_2;

// Rung 85: G1_GRAY_B1
// Binary bit = binary bit lebih tinggi XOR Gray bit
  LD %M102                (* G1_BIN_B2 *)
  XOR %M321               (* SIM_I1_1 *)
  ST %M101                (* G1_BIN_B1 *)
  // as ST:
  //   G1_BIN_B1 := G1_BIN_B2 XOR SIM_I1_1;

// Rung 86: G1_GRAY_B0
// Binary bit = binary bit lebih tinggi XOR Gray bit
  LD %M101                (* G1_BIN_B1 *)
  XOR %M320               (* SIM_I1_0 *)
  ST %M100                (* G1_BIN_B0 *)
  // as ST:
  //   G1_BIN_B0 := G1_BIN_B1 XOR SIM_I1_0;

// Rung 87: G1_BIN_CLEAR
// Mulai packing nilai biner
  LD 1
  [ %MW30 := 0 ]          (* ENC_BINARY_G1 *)
  // as ST:
  //   ENC_BINARY_G1 := 0;

// Rung 88: G1_BIN_ADD_1
// Tambahkan bobot bit yang aktif
  LD %M100                (* G1_BIN_B0 *)
  [ %MW30 := %MW30 + 1 ]  (* ENC_BINARY_G1, ENC_BINARY_G1 *)
  // as ST:
  //   IF G1_BIN_B0 THEN ENC_BINARY_G1 := ENC_BINARY_G1 + 1; END_IF;

// Rung 89: G1_BIN_ADD_2
// Tambahkan bobot bit yang aktif
  LD %M101                (* G1_BIN_B1 *)
  [ %MW30 := %MW30 + 2 ]  (* ENC_BINARY_G1, ENC_BINARY_G1 *)
  // as ST:
  //   IF G1_BIN_B1 THEN ENC_BINARY_G1 := ENC_BINARY_G1 + 2; END_IF;

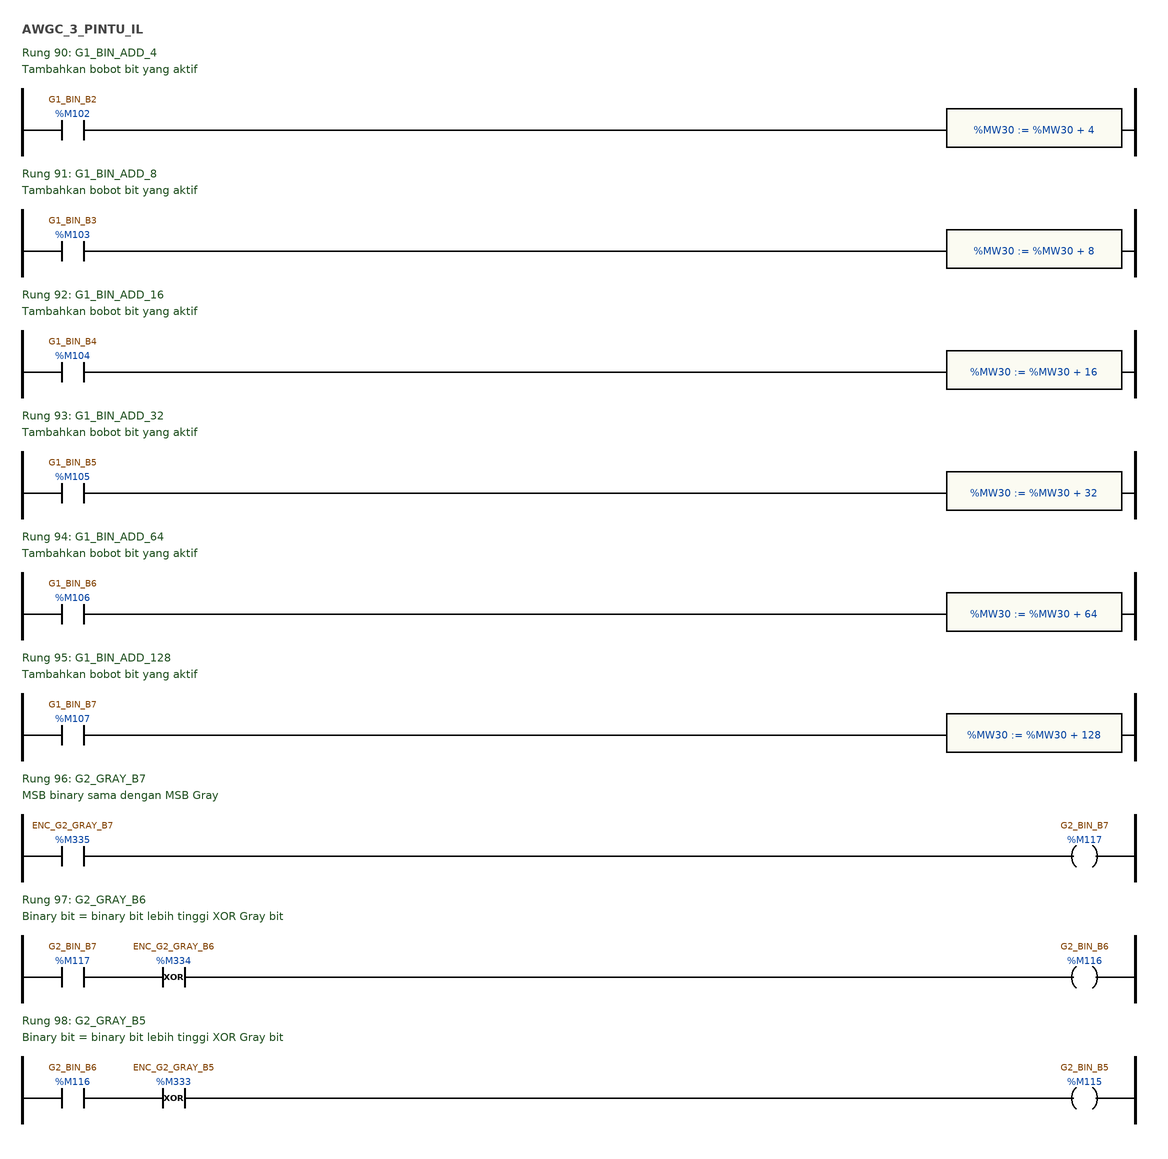

// Rung 90: G1_BIN_ADD_4
// Tambahkan bobot bit yang aktif
  LD %M102                (* G1_BIN_B2 *)
  [ %MW30 := %MW30 + 4 ]  (* ENC_BINARY_G1, ENC_BINARY_G1 *)
  // as ST:
  //   IF G1_BIN_B2 THEN ENC_BINARY_G1 := ENC_BINARY_G1 + 4; END_IF;

// Rung 91: G1_BIN_ADD_8
// Tambahkan bobot bit yang aktif
  LD %M103                (* G1_BIN_B3 *)
  [ %MW30 := %MW30 + 8 ]  (* ENC_BINARY_G1, ENC_BINARY_G1 *)
  // as ST:
  //   IF G1_BIN_B3 THEN ENC_BINARY_G1 := ENC_BINARY_G1 + 8; END_IF;

// Rung 92: G1_BIN_ADD_16
// Tambahkan bobot bit yang aktif
  LD %M104                (* G1_BIN_B4 *)
  [ %MW30 := %MW30 + 16 ] (* ENC_BINARY_G1, ENC_BINARY_G1 *)
  // as ST:
  //   IF G1_BIN_B4 THEN ENC_BINARY_G1 := ENC_BINARY_G1 + 16; END_IF;

// Rung 93: G1_BIN_ADD_32
// Tambahkan bobot bit yang aktif
  LD %M105                (* G1_BIN_B5 *)
  [ %MW30 := %MW30 + 32 ] (* ENC_BINARY_G1, ENC_BINARY_G1 *)
  // as ST:
  //   IF G1_BIN_B5 THEN ENC_BINARY_G1 := ENC_BINARY_G1 + 32; END_IF;

// Rung 94: G1_BIN_ADD_64
// Tambahkan bobot bit yang aktif
  LD %M106                (* G1_BIN_B6 *)
  [ %MW30 := %MW30 + 64 ] (* ENC_BINARY_G1, ENC_BINARY_G1 *)
  // as ST:
  //   IF G1_BIN_B6 THEN ENC_BINARY_G1 := ENC_BINARY_G1 + 64; END_IF;

// Rung 95: G1_BIN_ADD_128
// Tambahkan bobot bit yang aktif
  LD %M107                (* G1_BIN_B7 *)
  [ %MW30 := %MW30 + 128 ](* ENC_BINARY_G1, ENC_BINARY_G1 *)
  // as ST:
  //   IF G1_BIN_B7 THEN ENC_BINARY_G1 := ENC_BINARY_G1 + 128; END_IF;

// Rung 96: G2_GRAY_B7
// MSB binary sama dengan MSB Gray
  LD %M335                (* SIM_I1_15 *)
  ST %M117                (* G2_BIN_B7 *)
  // as ST:
  //   G2_BIN_B7 := SIM_I1_15;

// Rung 97: G2_GRAY_B6
// Binary bit = binary bit lebih tinggi XOR Gray bit
  LD %M117                (* G2_BIN_B7 *)
  XOR %M334               (* SIM_I1_14 *)
  ST %M116                (* G2_BIN_B6 *)
  // as ST:
  //   G2_BIN_B6 := G2_BIN_B7 XOR SIM_I1_14;

// Rung 98: G2_GRAY_B5
// Binary bit = binary bit lebih tinggi XOR Gray bit
  LD %M116                (* G2_BIN_B6 *)
  XOR %M333               (* SIM_I1_13 *)
  ST %M115                (* G2_BIN_B5 *)
  // as ST:
  //   G2_BIN_B5 := G2_BIN_B6 XOR SIM_I1_13;

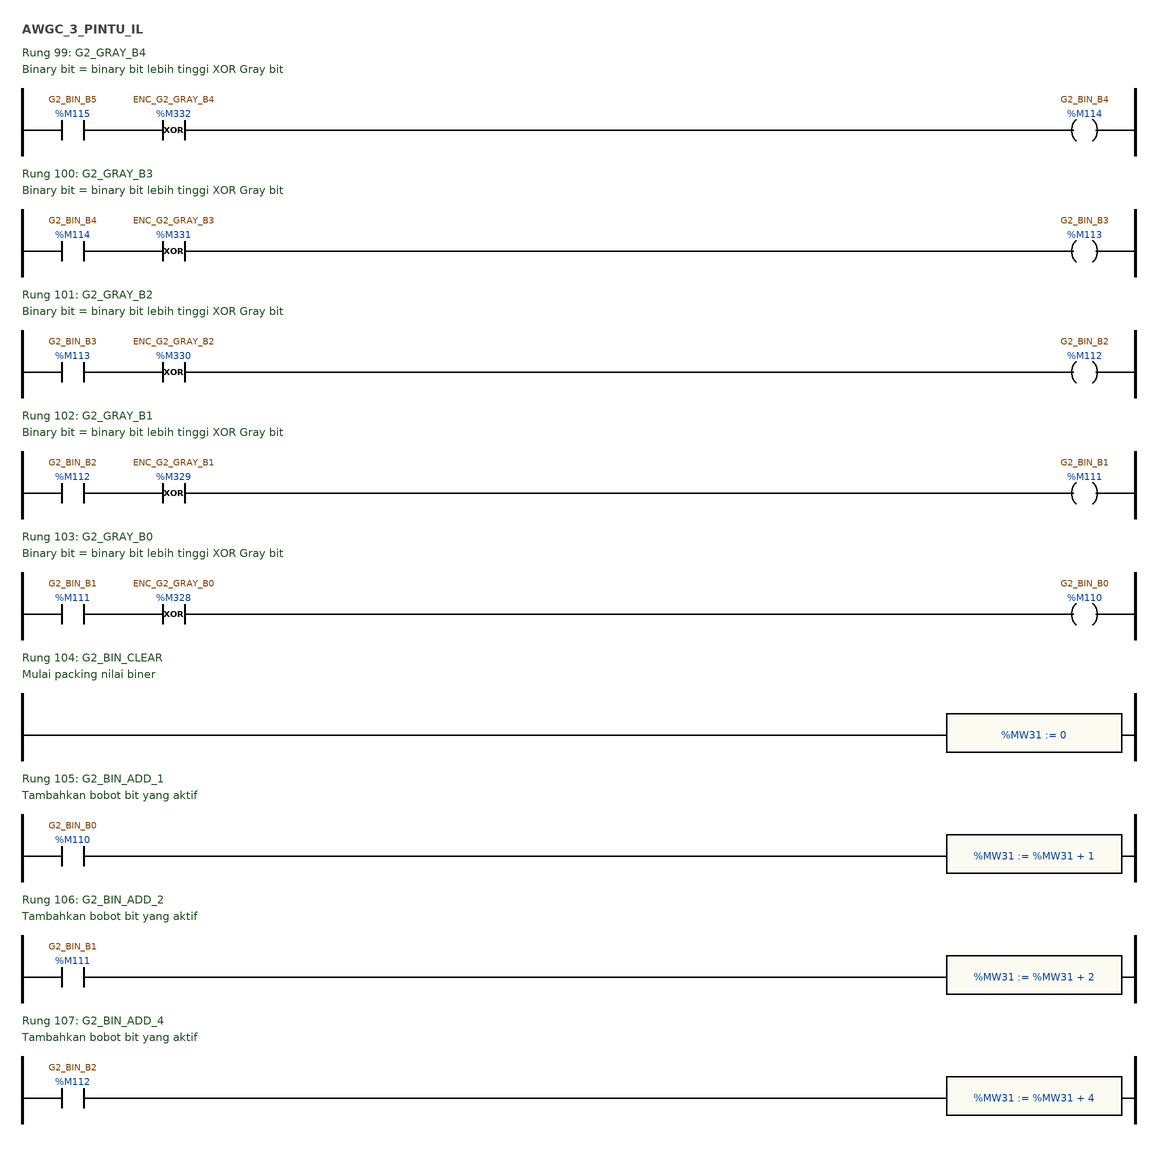

// Rung 99: G2_GRAY_B4
// Binary bit = binary bit lebih tinggi XOR Gray bit
  LD %M115                (* G2_BIN_B5 *)
  XOR %M332               (* SIM_I1_12 *)
  ST %M114                (* G2_BIN_B4 *)
  // as ST:
  //   G2_BIN_B4 := G2_BIN_B5 XOR SIM_I1_12;

// Rung 100: G2_GRAY_B3
// Binary bit = binary bit lebih tinggi XOR Gray bit
  LD %M114                (* G2_BIN_B4 *)
  XOR %M331               (* SIM_I1_11 *)
  ST %M113                (* G2_BIN_B3 *)
  // as ST:
  //   G2_BIN_B3 := G2_BIN_B4 XOR SIM_I1_11;

// Rung 101: G2_GRAY_B2
// Binary bit = binary bit lebih tinggi XOR Gray bit
  LD %M113                (* G2_BIN_B3 *)
  XOR %M330               (* SIM_I1_10 *)
  ST %M112                (* G2_BIN_B2 *)
  // as ST:
  //   G2_BIN_B2 := G2_BIN_B3 XOR SIM_I1_10;

// Rung 102: G2_GRAY_B1
// Binary bit = binary bit lebih tinggi XOR Gray bit
  LD %M112                (* G2_BIN_B2 *)
  XOR %M329               (* SIM_I1_9 *)
  ST %M111                (* G2_BIN_B1 *)
  // as ST:
  //   G2_BIN_B1 := G2_BIN_B2 XOR SIM_I1_9;

// Rung 103: G2_GRAY_B0
// Binary bit = binary bit lebih tinggi XOR Gray bit
  LD %M111                (* G2_BIN_B1 *)
  XOR %M328               (* SIM_I1_8 *)
  ST %M110                (* G2_BIN_B0 *)
  // as ST:
  //   G2_BIN_B0 := G2_BIN_B1 XOR SIM_I1_8;

// Rung 104: G2_BIN_CLEAR
// Mulai packing nilai biner
  LD 1
  [ %MW31 := 0 ]          (* ENC_BINARY_G2 *)
  // as ST:
  //   ENC_BINARY_G2 := 0;

// Rung 105: G2_BIN_ADD_1
// Tambahkan bobot bit yang aktif
  LD %M110                (* G2_BIN_B0 *)
  [ %MW31 := %MW31 + 1 ]  (* ENC_BINARY_G2, ENC_BINARY_G2 *)
  // as ST:
  //   IF G2_BIN_B0 THEN ENC_BINARY_G2 := ENC_BINARY_G2 + 1; END_IF;

// Rung 106: G2_BIN_ADD_2
// Tambahkan bobot bit yang aktif
  LD %M111                (* G2_BIN_B1 *)
  [ %MW31 := %MW31 + 2 ]  (* ENC_BINARY_G2, ENC_BINARY_G2 *)
  // as ST:
  //   IF G2_BIN_B1 THEN ENC_BINARY_G2 := ENC_BINARY_G2 + 2; END_IF;

// Rung 107: G2_BIN_ADD_4
// Tambahkan bobot bit yang aktif
  LD %M112                (* G2_BIN_B2 *)
  [ %MW31 := %MW31 + 4 ]  (* ENC_BINARY_G2, ENC_BINARY_G2 *)
  // as ST:
  //   IF G2_BIN_B2 THEN ENC_BINARY_G2 := ENC_BINARY_G2 + 4; END_IF;

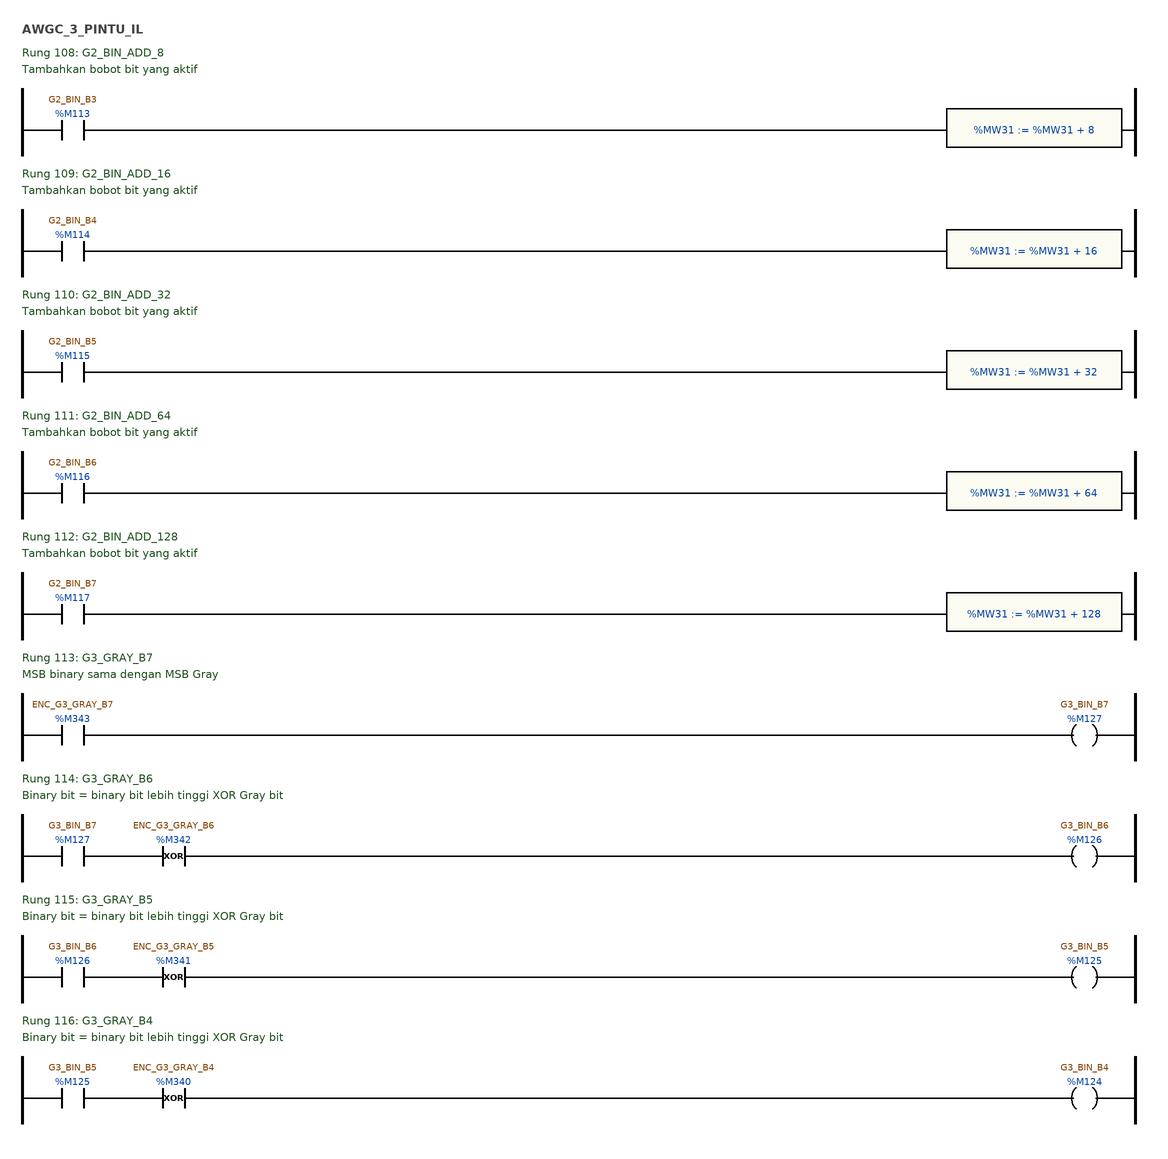

// Rung 108: G2_BIN_ADD_8
// Tambahkan bobot bit yang aktif
  LD %M113                (* G2_BIN_B3 *)
  [ %MW31 := %MW31 + 8 ]  (* ENC_BINARY_G2, ENC_BINARY_G2 *)
  // as ST:
  //   IF G2_BIN_B3 THEN ENC_BINARY_G2 := ENC_BINARY_G2 + 8; END_IF;

// Rung 109: G2_BIN_ADD_16
// Tambahkan bobot bit yang aktif
  LD %M114                (* G2_BIN_B4 *)
  [ %MW31 := %MW31 + 16 ] (* ENC_BINARY_G2, ENC_BINARY_G2 *)
  // as ST:
  //   IF G2_BIN_B4 THEN ENC_BINARY_G2 := ENC_BINARY_G2 + 16; END_IF;

// Rung 110: G2_BIN_ADD_32
// Tambahkan bobot bit yang aktif
  LD %M115                (* G2_BIN_B5 *)
  [ %MW31 := %MW31 + 32 ] (* ENC_BINARY_G2, ENC_BINARY_G2 *)
  // as ST:
  //   IF G2_BIN_B5 THEN ENC_BINARY_G2 := ENC_BINARY_G2 + 32; END_IF;

// Rung 111: G2_BIN_ADD_64
// Tambahkan bobot bit yang aktif
  LD %M116                (* G2_BIN_B6 *)
  [ %MW31 := %MW31 + 64 ] (* ENC_BINARY_G2, ENC_BINARY_G2 *)
  // as ST:
  //   IF G2_BIN_B6 THEN ENC_BINARY_G2 := ENC_BINARY_G2 + 64; END_IF;

// Rung 112: G2_BIN_ADD_128
// Tambahkan bobot bit yang aktif
  LD %M117                (* G2_BIN_B7 *)
  [ %MW31 := %MW31 + 128 ](* ENC_BINARY_G2, ENC_BINARY_G2 *)
  // as ST:
  //   IF G2_BIN_B7 THEN ENC_BINARY_G2 := ENC_BINARY_G2 + 128; END_IF;

// Rung 113: G3_GRAY_B7
// MSB binary sama dengan MSB Gray
  LD %M343                (* SIM_I1_23 *)
  ST %M127                (* G3_BIN_B7 *)
  // as ST:
  //   G3_BIN_B7 := SIM_I1_23;

// Rung 114: G3_GRAY_B6
// Binary bit = binary bit lebih tinggi XOR Gray bit
  LD %M127                (* G3_BIN_B7 *)
  XOR %M342               (* SIM_I1_22 *)
  ST %M126                (* G3_BIN_B6 *)
  // as ST:
  //   G3_BIN_B6 := G3_BIN_B7 XOR SIM_I1_22;

// Rung 115: G3_GRAY_B5
// Binary bit = binary bit lebih tinggi XOR Gray bit
  LD %M126                (* G3_BIN_B6 *)
  XOR %M341               (* SIM_I1_21 *)
  ST %M125                (* G3_BIN_B5 *)
  // as ST:
  //   G3_BIN_B5 := G3_BIN_B6 XOR SIM_I1_21;

// Rung 116: G3_GRAY_B4
// Binary bit = binary bit lebih tinggi XOR Gray bit
  LD %M125                (* G3_BIN_B5 *)
  XOR %M340               (* SIM_I1_20 *)
  ST %M124                (* G3_BIN_B4 *)
  // as ST:
  //   G3_BIN_B4 := G3_BIN_B5 XOR SIM_I1_20;

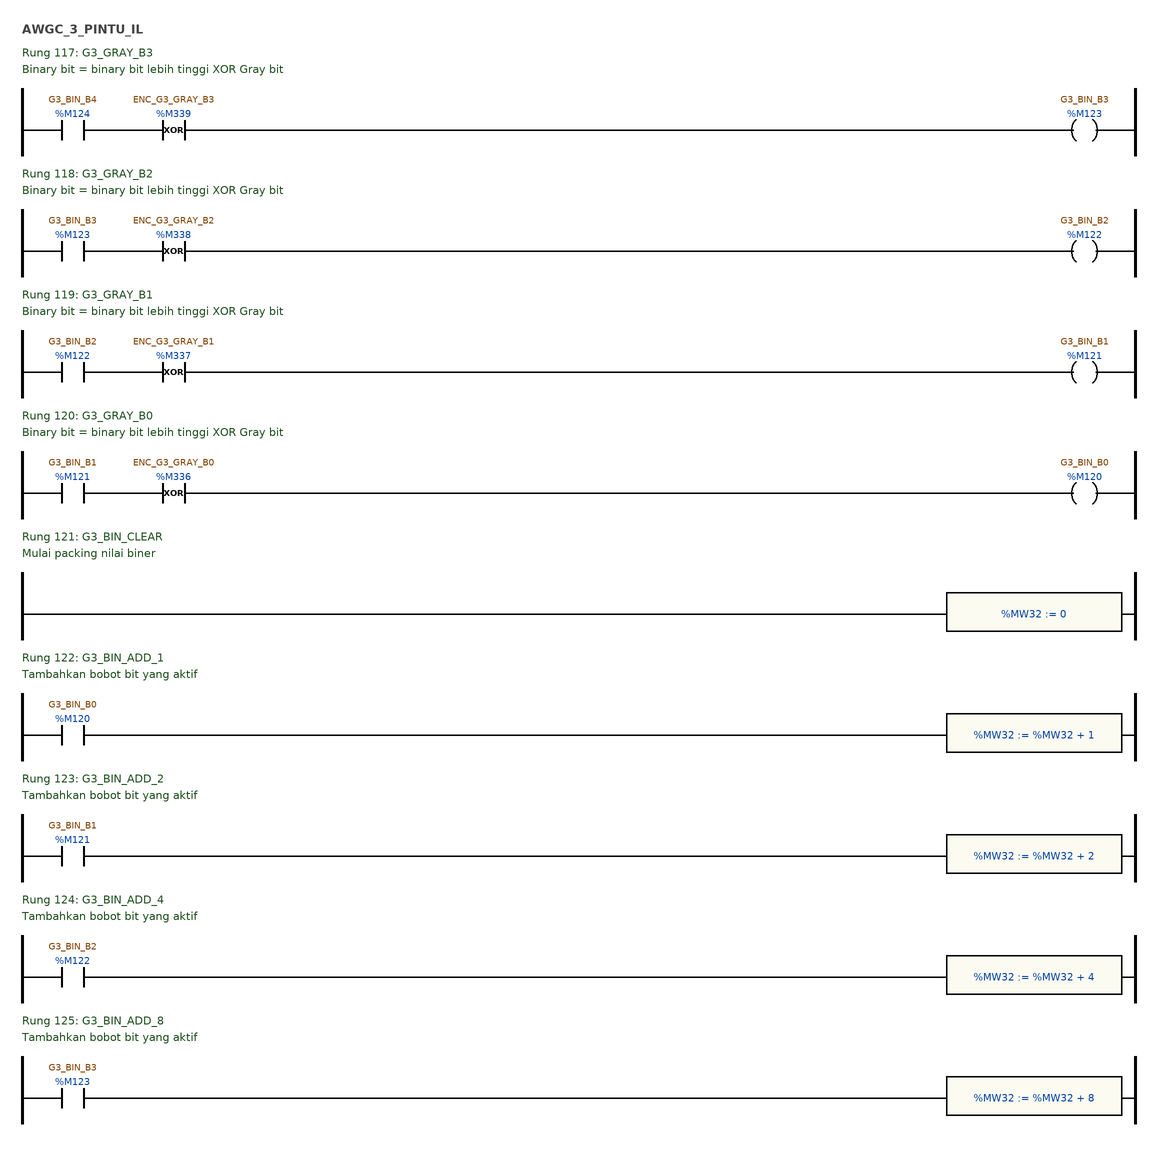

// Rung 117: G3_GRAY_B3
// Binary bit = binary bit lebih tinggi XOR Gray bit
  LD %M124                (* G3_BIN_B4 *)
  XOR %M339               (* SIM_I1_19 *)
  ST %M123                (* G3_BIN_B3 *)
  // as ST:
  //   G3_BIN_B3 := G3_BIN_B4 XOR SIM_I1_19;

// Rung 118: G3_GRAY_B2
// Binary bit = binary bit lebih tinggi XOR Gray bit
  LD %M123                (* G3_BIN_B3 *)
  XOR %M338               (* SIM_I1_18 *)
  ST %M122                (* G3_BIN_B2 *)
  // as ST:
  //   G3_BIN_B2 := G3_BIN_B3 XOR SIM_I1_18;

// Rung 119: G3_GRAY_B1
// Binary bit = binary bit lebih tinggi XOR Gray bit
  LD %M122                (* G3_BIN_B2 *)
  XOR %M337               (* SIM_I1_17 *)
  ST %M121                (* G3_BIN_B1 *)
  // as ST:
  //   G3_BIN_B1 := G3_BIN_B2 XOR SIM_I1_17;

// Rung 120: G3_GRAY_B0
// Binary bit = binary bit lebih tinggi XOR Gray bit
  LD %M121                (* G3_BIN_B1 *)
  XOR %M336               (* SIM_I1_16 *)
  ST %M120                (* G3_BIN_B0 *)
  // as ST:
  //   G3_BIN_B0 := G3_BIN_B1 XOR SIM_I1_16;

// Rung 121: G3_BIN_CLEAR
// Mulai packing nilai biner
  LD 1
  [ %MW32 := 0 ]          (* ENC_BINARY_G3 *)
  // as ST:
  //   ENC_BINARY_G3 := 0;

// Rung 122: G3_BIN_ADD_1
// Tambahkan bobot bit yang aktif
  LD %M120                (* G3_BIN_B0 *)
  [ %MW32 := %MW32 + 1 ]  (* ENC_BINARY_G3, ENC_BINARY_G3 *)
  // as ST:
  //   IF G3_BIN_B0 THEN ENC_BINARY_G3 := ENC_BINARY_G3 + 1; END_IF;

// Rung 123: G3_BIN_ADD_2
// Tambahkan bobot bit yang aktif
  LD %M121                (* G3_BIN_B1 *)
  [ %MW32 := %MW32 + 2 ]  (* ENC_BINARY_G3, ENC_BINARY_G3 *)
  // as ST:
  //   IF G3_BIN_B1 THEN ENC_BINARY_G3 := ENC_BINARY_G3 + 2; END_IF;

// Rung 124: G3_BIN_ADD_4
// Tambahkan bobot bit yang aktif
  LD %M122                (* G3_BIN_B2 *)
  [ %MW32 := %MW32 + 4 ]  (* ENC_BINARY_G3, ENC_BINARY_G3 *)
  // as ST:
  //   IF G3_BIN_B2 THEN ENC_BINARY_G3 := ENC_BINARY_G3 + 4; END_IF;

// Rung 125: G3_BIN_ADD_8
// Tambahkan bobot bit yang aktif
  LD %M123                (* G3_BIN_B3 *)
  [ %MW32 := %MW32 + 8 ]  (* ENC_BINARY_G3, ENC_BINARY_G3 *)
  // as ST:
  //   IF G3_BIN_B3 THEN ENC_BINARY_G3 := ENC_BINARY_G3 + 8; END_IF;

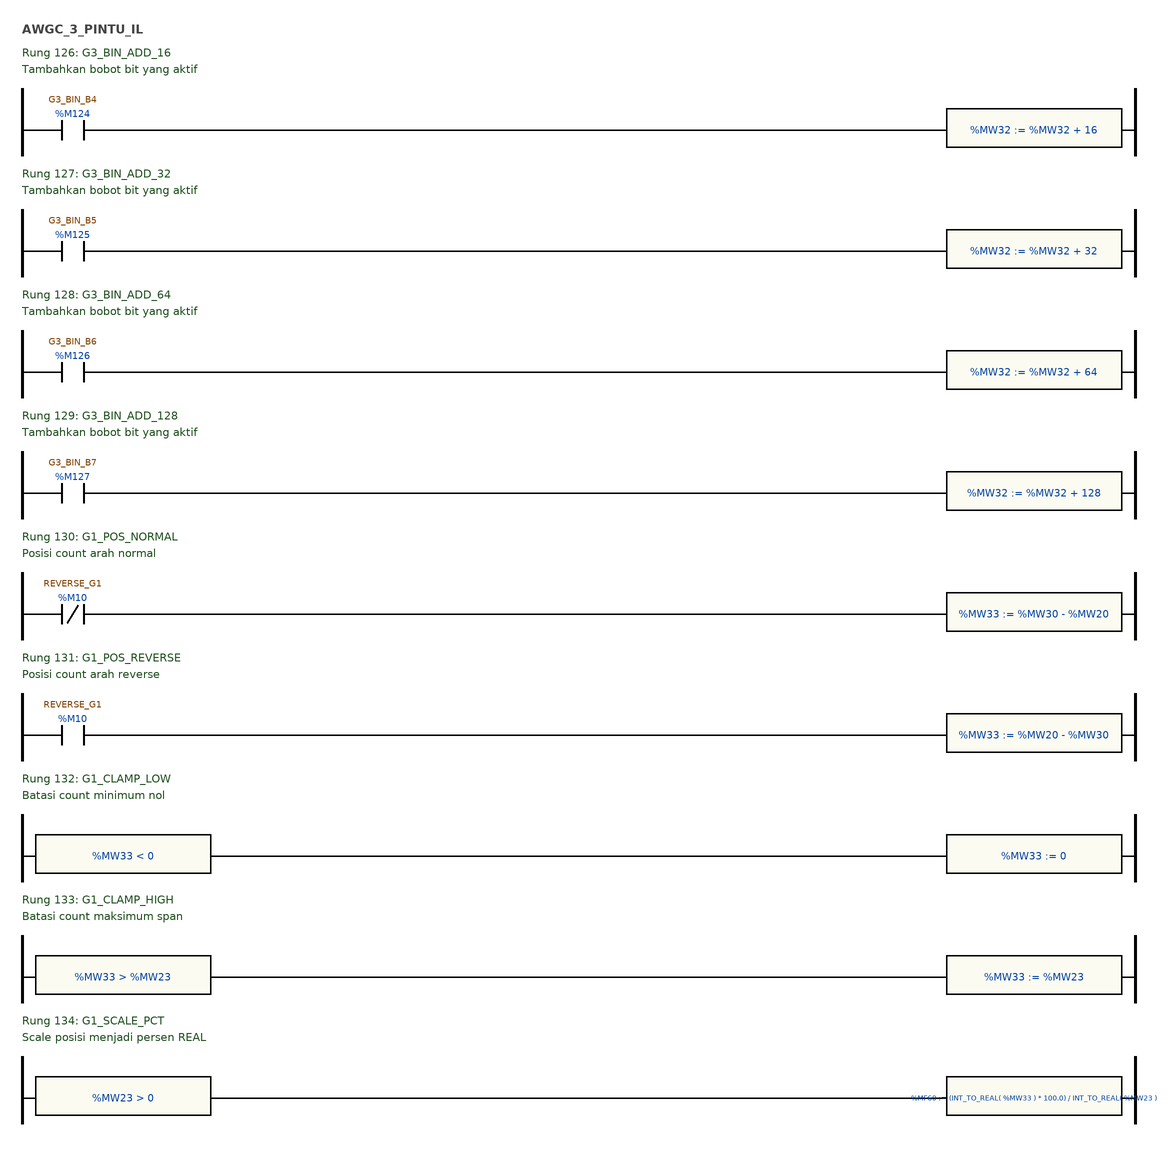

// Rung 126: G3_BIN_ADD_16
// Tambahkan bobot bit yang aktif
  LD %M124                (* G3_BIN_B4 *)
  [ %MW32 := %MW32 + 16 ] (* ENC_BINARY_G3, ENC_BINARY_G3 *)
  // as ST:
  //   IF G3_BIN_B4 THEN ENC_BINARY_G3 := ENC_BINARY_G3 + 16; END_IF;

// Rung 127: G3_BIN_ADD_32
// Tambahkan bobot bit yang aktif
  LD %M125                (* G3_BIN_B5 *)
  [ %MW32 := %MW32 + 32 ] (* ENC_BINARY_G3, ENC_BINARY_G3 *)
  // as ST:
  //   IF G3_BIN_B5 THEN ENC_BINARY_G3 := ENC_BINARY_G3 + 32; END_IF;

// Rung 128: G3_BIN_ADD_64
// Tambahkan bobot bit yang aktif
  LD %M126                (* G3_BIN_B6 *)
  [ %MW32 := %MW32 + 64 ] (* ENC_BINARY_G3, ENC_BINARY_G3 *)
  // as ST:
  //   IF G3_BIN_B6 THEN ENC_BINARY_G3 := ENC_BINARY_G3 + 64; END_IF;

// Rung 129: G3_BIN_ADD_128
// Tambahkan bobot bit yang aktif
  LD %M127                (* G3_BIN_B7 *)
  [ %MW32 := %MW32 + 128 ](* ENC_BINARY_G3, ENC_BINARY_G3 *)
  // as ST:
  //   IF G3_BIN_B7 THEN ENC_BINARY_G3 := ENC_BINARY_G3 + 128; END_IF;

// Rung 130: G1_POS_NORMAL
// Posisi count arah normal
  LDN %M10                (* REVERSE_G1 *)
  [ %MW33 := %MW30 - %MW20 ](* POS_COUNT_G1, ENC_BINARY_G1, ENC_ZERO_G1 *)
  // as ST:
  //   IF NOT REVERSE_G1 THEN POS_COUNT_G1 := ENC_BINARY_G1 - ENC_ZERO_G1; END_IF;

// Rung 131: G1_POS_REVERSE
// Posisi count arah reverse
  LD %M10                 (* REVERSE_G1 *)
  [ %MW33 := %MW20 - %MW30 ](* POS_COUNT_G1, ENC_ZERO_G1, ENC_BINARY_G1 *)
  // as ST:
  //   IF REVERSE_G1 THEN POS_COUNT_G1 := ENC_ZERO_G1 - ENC_BINARY_G1; END_IF;

// Rung 132: G1_CLAMP_LOW
// Batasi count minimum nol
  LD [ %MW33 < 0 ]        (* POS_COUNT_G1 *)
  [ %MW33 := 0 ]          (* POS_COUNT_G1 *)
  // as ST:
  //   IF POS_COUNT_G1 < 0 THEN POS_COUNT_G1 := 0; END_IF;

// Rung 133: G1_CLAMP_HIGH
// Batasi count maksimum span
  LD [ %MW33 > %MW23 ]    (* POS_COUNT_G1, ENC_SPAN_G1 *)
  [ %MW33 := %MW23 ]      (* POS_COUNT_G1, ENC_SPAN_G1 *)
  // as ST:
  //   IF POS_COUNT_G1 > ENC_SPAN_G1 THEN POS_COUNT_G1 := ENC_SPAN_G1; END_IF;

// Rung 134: G1_SCALE_PCT
// Scale posisi menjadi persen REAL
  LD [ %MW23 > 0 ]        (* ENC_SPAN_G1 *)
  [ %MF60 := ( INT_TO_REAL ( %MW33 ) * 100.0 ) / INT_TO_REAL ( %MW23 ) ](* POSITION_G1_PCT, POS_COUNT_G1, ENC_SPAN_G1 *)
  // as ST:
  //   IF ENC_SPAN_G1 > 0 THEN POSITION_G1_PCT := ( INT_TO_REAL ( POS_COUNT_G1 ) * 100.0 ) / INT_TO_REAL ( ENC_SPAN_G1 ); END_IF;

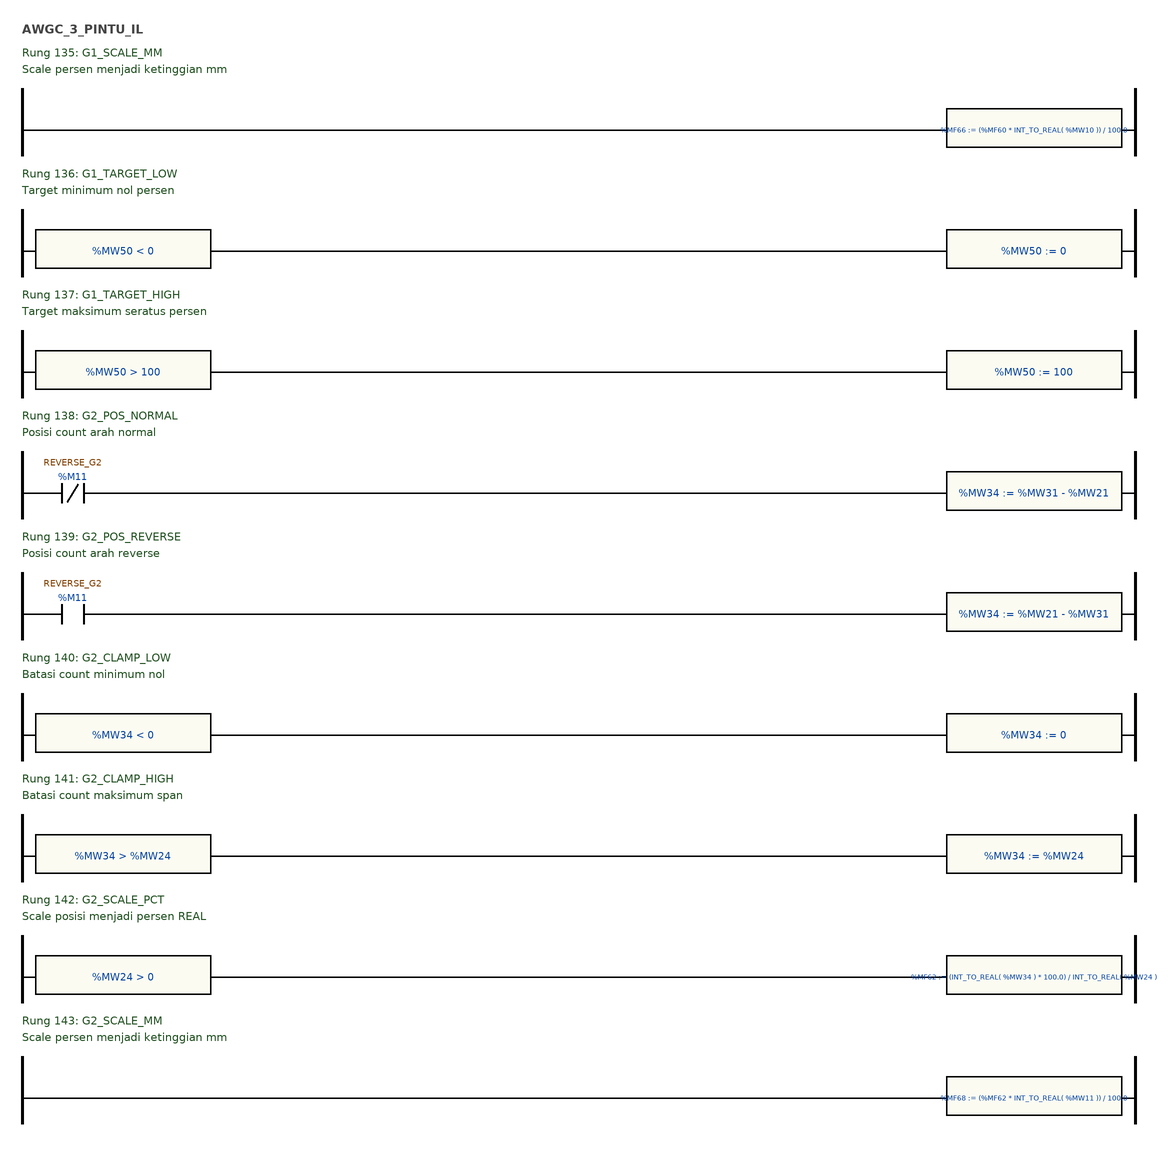

// Rung 135: G1_SCALE_MM
// Scale persen menjadi ketinggian mm
  LD 1
  [ %MF66 := ( %MF60 * INT_TO_REAL ( %MW10 ) ) / 100.0 ](* POSITION_G1_MM, POSITION_G1_PCT, MAX_HEIGHT_G1_MM *)
  // as ST:
  //   POSITION_G1_MM := ( POSITION_G1_PCT * INT_TO_REAL ( MAX_HEIGHT_G1_MM ) ) / 100.0;

// Rung 136: G1_TARGET_LOW
// Target minimum nol persen
  LD [ %MW50 < 0 ]        (* TARGET_PCT_G1 *)
  [ %MW50 := 0 ]          (* TARGET_PCT_G1 *)
  // as ST:
  //   IF TARGET_PCT_G1 < 0 THEN TARGET_PCT_G1 := 0; END_IF;

// Rung 137: G1_TARGET_HIGH
// Target maksimum seratus persen
  LD [ %MW50 > 100 ]      (* TARGET_PCT_G1 *)
  [ %MW50 := 100 ]        (* TARGET_PCT_G1 *)
  // as ST:
  //   IF TARGET_PCT_G1 > 100 THEN TARGET_PCT_G1 := 100; END_IF;

// Rung 138: G2_POS_NORMAL
// Posisi count arah normal
  LDN %M11                (* REVERSE_G2 *)
  [ %MW34 := %MW31 - %MW21 ](* POS_COUNT_G2, ENC_BINARY_G2, ENC_ZERO_G2 *)
  // as ST:
  //   IF NOT REVERSE_G2 THEN POS_COUNT_G2 := ENC_BINARY_G2 - ENC_ZERO_G2; END_IF;

// Rung 139: G2_POS_REVERSE
// Posisi count arah reverse
  LD %M11                 (* REVERSE_G2 *)
  [ %MW34 := %MW21 - %MW31 ](* POS_COUNT_G2, ENC_ZERO_G2, ENC_BINARY_G2 *)
  // as ST:
  //   IF REVERSE_G2 THEN POS_COUNT_G2 := ENC_ZERO_G2 - ENC_BINARY_G2; END_IF;

// Rung 140: G2_CLAMP_LOW
// Batasi count minimum nol
  LD [ %MW34 < 0 ]        (* POS_COUNT_G2 *)
  [ %MW34 := 0 ]          (* POS_COUNT_G2 *)
  // as ST:
  //   IF POS_COUNT_G2 < 0 THEN POS_COUNT_G2 := 0; END_IF;

// Rung 141: G2_CLAMP_HIGH
// Batasi count maksimum span
  LD [ %MW34 > %MW24 ]    (* POS_COUNT_G2, ENC_SPAN_G2 *)
  [ %MW34 := %MW24 ]      (* POS_COUNT_G2, ENC_SPAN_G2 *)
  // as ST:
  //   IF POS_COUNT_G2 > ENC_SPAN_G2 THEN POS_COUNT_G2 := ENC_SPAN_G2; END_IF;

// Rung 142: G2_SCALE_PCT
// Scale posisi menjadi persen REAL
  LD [ %MW24 > 0 ]        (* ENC_SPAN_G2 *)
  [ %MF62 := ( INT_TO_REAL ( %MW34 ) * 100.0 ) / INT_TO_REAL ( %MW24 ) ](* POSITION_G2_PCT, POS_COUNT_G2, ENC_SPAN_G2 *)
  // as ST:
  //   IF ENC_SPAN_G2 > 0 THEN POSITION_G2_PCT := ( INT_TO_REAL ( POS_COUNT_G2 ) * 100.0 ) / INT_TO_REAL ( ENC_SPAN_G2 ); END_IF;

// Rung 143: G2_SCALE_MM
// Scale persen menjadi ketinggian mm
  LD 1
  [ %MF68 := ( %MF62 * INT_TO_REAL ( %MW11 ) ) / 100.0 ](* POSITION_G2_MM, POSITION_G2_PCT, MAX_HEIGHT_G2_MM *)
  // as ST:
  //   POSITION_G2_MM := ( POSITION_G2_PCT * INT_TO_REAL ( MAX_HEIGHT_G2_MM ) ) / 100.0;

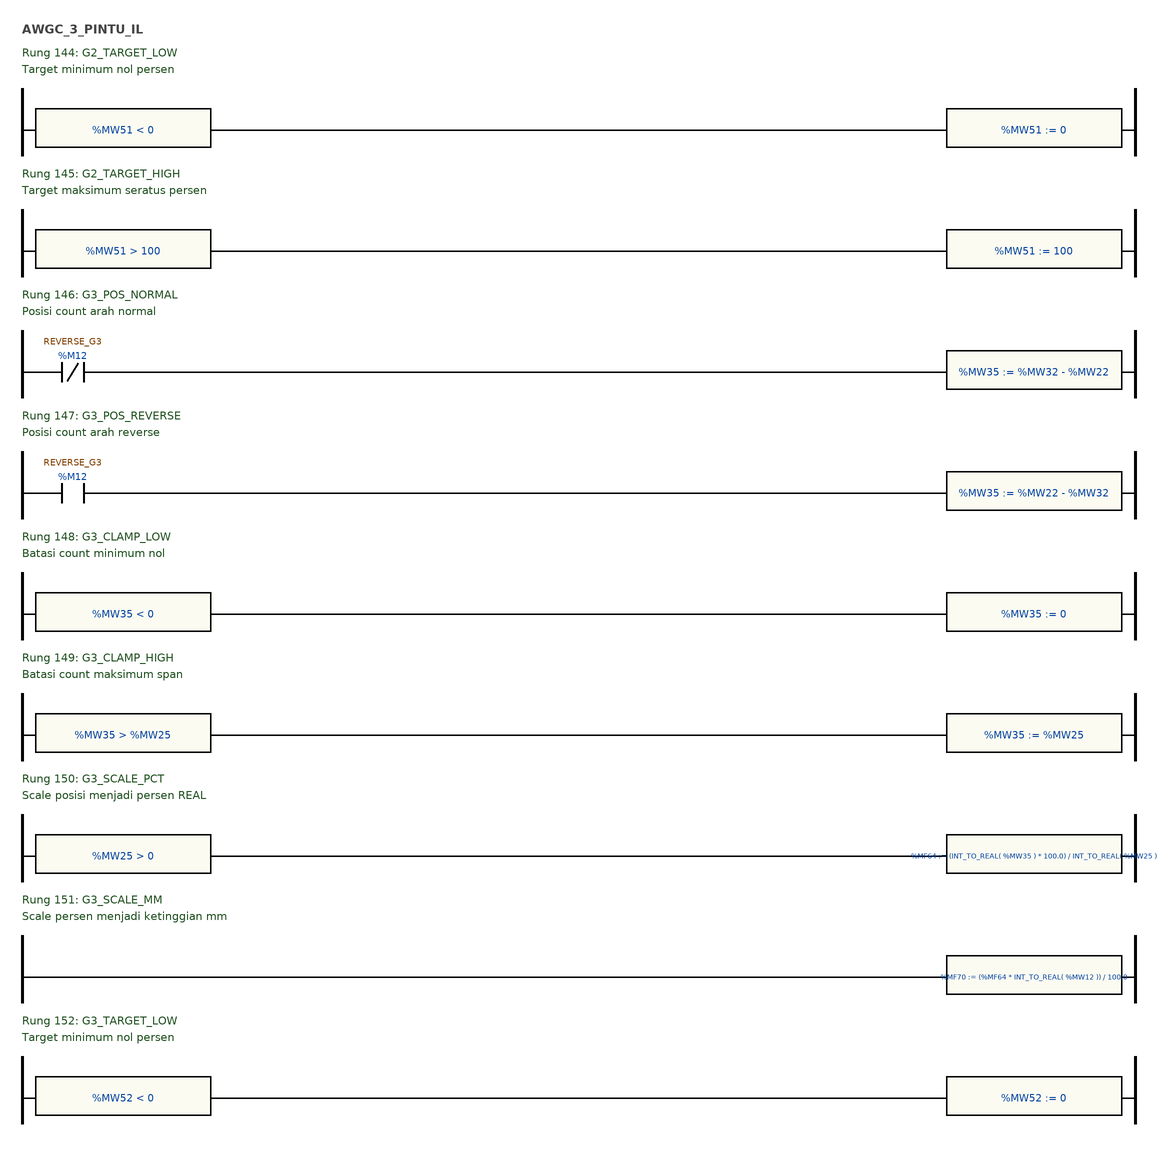

// Rung 144: G2_TARGET_LOW
// Target minimum nol persen
  LD [ %MW51 < 0 ]        (* TARGET_PCT_G2 *)
  [ %MW51 := 0 ]          (* TARGET_PCT_G2 *)
  // as ST:
  //   IF TARGET_PCT_G2 < 0 THEN TARGET_PCT_G2 := 0; END_IF;

// Rung 145: G2_TARGET_HIGH
// Target maksimum seratus persen
  LD [ %MW51 > 100 ]      (* TARGET_PCT_G2 *)
  [ %MW51 := 100 ]        (* TARGET_PCT_G2 *)
  // as ST:
  //   IF TARGET_PCT_G2 > 100 THEN TARGET_PCT_G2 := 100; END_IF;

// Rung 146: G3_POS_NORMAL
// Posisi count arah normal
  LDN %M12                (* REVERSE_G3 *)
  [ %MW35 := %MW32 - %MW22 ](* POS_COUNT_G3, ENC_BINARY_G3, ENC_ZERO_G3 *)
  // as ST:
  //   IF NOT REVERSE_G3 THEN POS_COUNT_G3 := ENC_BINARY_G3 - ENC_ZERO_G3; END_IF;

// Rung 147: G3_POS_REVERSE
// Posisi count arah reverse
  LD %M12                 (* REVERSE_G3 *)
  [ %MW35 := %MW22 - %MW32 ](* POS_COUNT_G3, ENC_ZERO_G3, ENC_BINARY_G3 *)
  // as ST:
  //   IF REVERSE_G3 THEN POS_COUNT_G3 := ENC_ZERO_G3 - ENC_BINARY_G3; END_IF;

// Rung 148: G3_CLAMP_LOW
// Batasi count minimum nol
  LD [ %MW35 < 0 ]        (* POS_COUNT_G3 *)
  [ %MW35 := 0 ]          (* POS_COUNT_G3 *)
  // as ST:
  //   IF POS_COUNT_G3 < 0 THEN POS_COUNT_G3 := 0; END_IF;

// Rung 149: G3_CLAMP_HIGH
// Batasi count maksimum span
  LD [ %MW35 > %MW25 ]    (* POS_COUNT_G3, ENC_SPAN_G3 *)
  [ %MW35 := %MW25 ]      (* POS_COUNT_G3, ENC_SPAN_G3 *)
  // as ST:
  //   IF POS_COUNT_G3 > ENC_SPAN_G3 THEN POS_COUNT_G3 := ENC_SPAN_G3; END_IF;

// Rung 150: G3_SCALE_PCT
// Scale posisi menjadi persen REAL
  LD [ %MW25 > 0 ]        (* ENC_SPAN_G3 *)
  [ %MF64 := ( INT_TO_REAL ( %MW35 ) * 100.0 ) / INT_TO_REAL ( %MW25 ) ](* POSITION_G3_PCT, POS_COUNT_G3, ENC_SPAN_G3 *)
  // as ST:
  //   IF ENC_SPAN_G3 > 0 THEN POSITION_G3_PCT := ( INT_TO_REAL ( POS_COUNT_G3 ) * 100.0 ) / INT_TO_REAL ( ENC_SPAN_G3 ); END_IF;

// Rung 151: G3_SCALE_MM
// Scale persen menjadi ketinggian mm
  LD 1
  [ %MF70 := ( %MF64 * INT_TO_REAL ( %MW12 ) ) / 100.0 ](* POSITION_G3_MM, POSITION_G3_PCT, MAX_HEIGHT_G3_MM *)
  // as ST:
  //   POSITION_G3_MM := ( POSITION_G3_PCT * INT_TO_REAL ( MAX_HEIGHT_G3_MM ) ) / 100.0;

// Rung 152: G3_TARGET_LOW
// Target minimum nol persen
  LD [ %MW52 < 0 ]        (* TARGET_PCT_G3 *)
  [ %MW52 := 0 ]          (* TARGET_PCT_G3 *)
  // as ST:
  //   IF TARGET_PCT_G3 < 0 THEN TARGET_PCT_G3 := 0; END_IF;

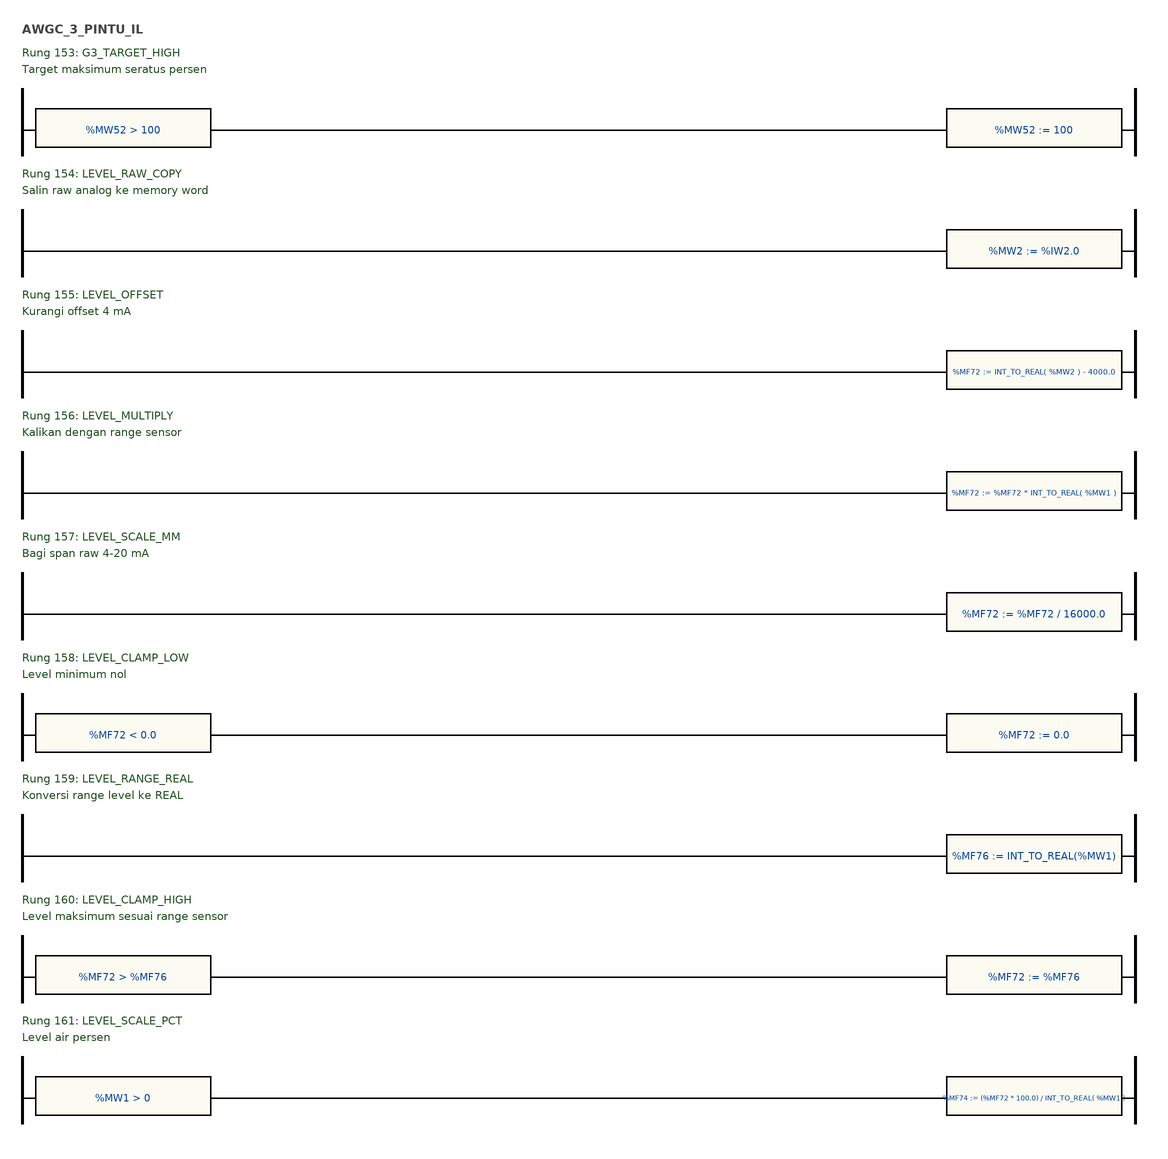

// Rung 153: G3_TARGET_HIGH
// Target maksimum seratus persen
  LD [ %MW52 > 100 ]      (* TARGET_PCT_G3 *)
  [ %MW52 := 100 ]        (* TARGET_PCT_G3 *)
  // as ST:
  //   IF TARGET_PCT_G3 > 100 THEN TARGET_PCT_G3 := 100; END_IF;

// Rung 154: LEVEL_RAW_COPY
// Salin raw analog ke memory word
  LD 1
  [ %MW2 := %IW2.0 ]      (* LEVEL_RAW_COPY, LEVEL_RAW *)
  // as ST:
  //   LEVEL_RAW_COPY := LEVEL_RAW;

// Rung 155: LEVEL_OFFSET
// Kurangi offset 4 mA
  LD 1
  [ %MF72 := INT_TO_REAL ( %MW2 ) - 4000.0 ](* WATER_LEVEL_MM, LEVEL_RAW_COPY *)
  // as ST:
  //   WATER_LEVEL_MM := INT_TO_REAL ( LEVEL_RAW_COPY ) - 4000.0;

// Rung 156: LEVEL_MULTIPLY
// Kalikan dengan range sensor
  LD 1
  [ %MF72 := %MF72 * INT_TO_REAL ( %MW1 ) ](* WATER_LEVEL_MM, WATER_LEVEL_MM, WATER_RANGE_MM *)
  // as ST:
  //   WATER_LEVEL_MM := WATER_LEVEL_MM * INT_TO_REAL ( WATER_RANGE_MM );

// Rung 157: LEVEL_SCALE_MM
// Bagi span raw 4-20 mA
  LD 1
  [ %MF72 := %MF72 / 16000.0 ](* WATER_LEVEL_MM, WATER_LEVEL_MM *)
  // as ST:
  //   WATER_LEVEL_MM := WATER_LEVEL_MM / 16000.0;

// Rung 158: LEVEL_CLAMP_LOW
// Level minimum nol
  LD [ %MF72 < 0.0 ]      (* WATER_LEVEL_MM *)
  [ %MF72 := 0.0 ]        (* WATER_LEVEL_MM *)
  // as ST:
  //   IF WATER_LEVEL_MM < 0.0 THEN WATER_LEVEL_MM := 0.0; END_IF;

// Rung 159: LEVEL_RANGE_REAL
// Konversi range level ke REAL
  LD 1
  [ %MF76 := INT_TO_REAL ( %MW1 ) ](* WATER_RANGE_REAL, WATER_RANGE_MM *)
  // as ST:
  //   WATER_RANGE_REAL := INT_TO_REAL ( WATER_RANGE_MM );

// Rung 160: LEVEL_CLAMP_HIGH
// Level maksimum sesuai range sensor
  LD [ %MF72 > %MF76 ]    (* WATER_LEVEL_MM, WATER_RANGE_REAL *)
  [ %MF72 := %MF76 ]      (* WATER_LEVEL_MM, WATER_RANGE_REAL *)
  // as ST:
  //   IF WATER_LEVEL_MM > WATER_RANGE_REAL THEN WATER_LEVEL_MM := WATER_RANGE_REAL; END_IF;

// Rung 161: LEVEL_SCALE_PCT
// Level air persen
  LD [ %MW1 > 0 ]         (* WATER_RANGE_MM *)
  [ %MF74 := ( %MF72 * 100.0 ) / INT_TO_REAL ( %MW1 ) ](* WATER_LEVEL_PCT, WATER_LEVEL_MM, WATER_RANGE_MM *)
  // as ST:
  //   IF WATER_RANGE_MM > 0 THEN WATER_LEVEL_PCT := ( WATER_LEVEL_MM * 100.0 ) / INT_TO_REAL ( WATER_RANGE_MM ); END_IF;

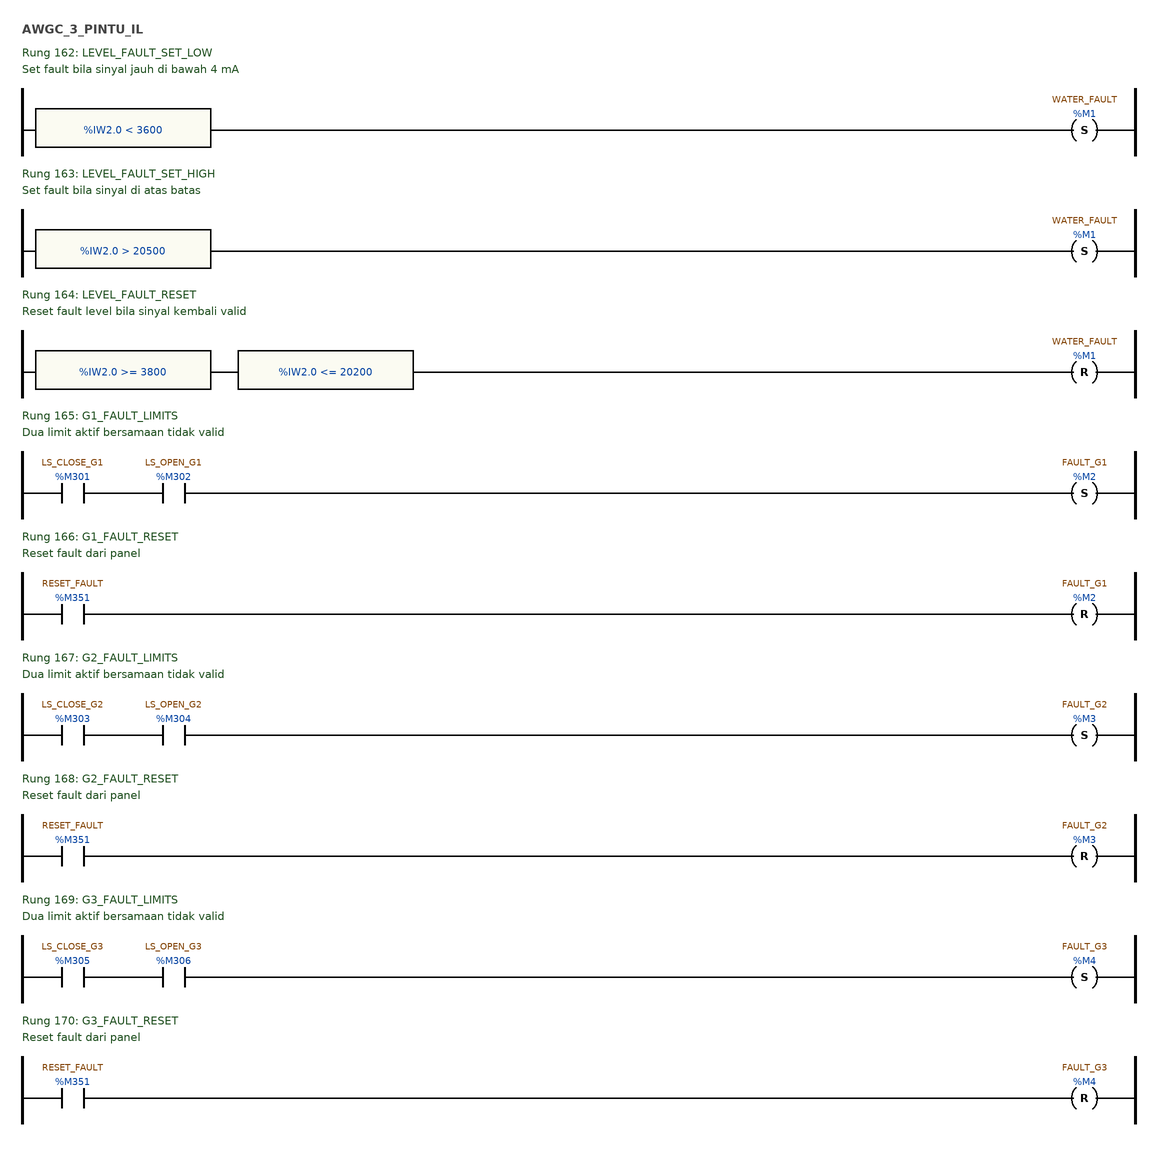

// Rung 162: LEVEL_FAULT_SET_LOW
// Set fault bila sinyal jauh di bawah 4 mA
  LD [ %IW2.0 < 3600 ]    (* LEVEL_RAW *)
  S %M1                   (* WATER_FAULT *)
  // as ST:
  //   IF LEVEL_RAW < 3600 THEN WATER_FAULT := TRUE; END_IF;

// Rung 163: LEVEL_FAULT_SET_HIGH
// Set fault bila sinyal di atas batas
  LD [ %IW2.0 > 20500 ]   (* LEVEL_RAW *)
  S %M1                   (* WATER_FAULT *)
  // as ST:
  //   IF LEVEL_RAW > 20500 THEN WATER_FAULT := TRUE; END_IF;

// Rung 164: LEVEL_FAULT_RESET
// Reset fault level bila sinyal kembali valid
  LD [ %IW2.0 >= 3800 ]   (* LEVEL_RAW *)
  AND [ %IW2.0 <= 20200 ] (* LEVEL_RAW *)
  R %M1                   (* WATER_FAULT *)
  // as ST:
  //   IF LEVEL_RAW >= 3800 AND LEVEL_RAW <= 20200 THEN WATER_FAULT := FALSE; END_IF;

// Rung 165: G1_FAULT_LIMITS
// Dua limit aktif bersamaan tidak valid
  LD %M301                (* SCADA_LS_CLOSE_G1 *)
  AND %M302               (* SCADA_LS_OPEN_G1 *)
  S %M2                   (* FAULT_G1 *)
  // as ST:
  //   IF SCADA_LS_CLOSE_G1 AND SCADA_LS_OPEN_G1 THEN FAULT_G1 := TRUE; END_IF;

// Rung 166: G1_FAULT_RESET
// Reset fault dari panel
  LD %M351                (* SCADA_RESET_FAULT *)
  R %M2                   (* FAULT_G1 *)
  // as ST:
  //   IF SCADA_RESET_FAULT THEN FAULT_G1 := FALSE; END_IF;

// Rung 167: G2_FAULT_LIMITS
// Dua limit aktif bersamaan tidak valid
  LD %M303                (* SCADA_LS_CLOSE_G2 *)
  AND %M304               (* SCADA_LS_OPEN_G2 *)
  S %M3                   (* FAULT_G2 *)
  // as ST:
  //   IF SCADA_LS_CLOSE_G2 AND SCADA_LS_OPEN_G2 THEN FAULT_G2 := TRUE; END_IF;

// Rung 168: G2_FAULT_RESET
// Reset fault dari panel
  LD %M351                (* SCADA_RESET_FAULT *)
  R %M3                   (* FAULT_G2 *)
  // as ST:
  //   IF SCADA_RESET_FAULT THEN FAULT_G2 := FALSE; END_IF;

// Rung 169: G3_FAULT_LIMITS
// Dua limit aktif bersamaan tidak valid
  LD %M305                (* SCADA_LS_CLOSE_G3 *)
  AND %M306               (* SCADA_LS_OPEN_G3 *)
  S %M4                   (* FAULT_G3 *)
  // as ST:
  //   IF SCADA_LS_CLOSE_G3 AND SCADA_LS_OPEN_G3 THEN FAULT_G3 := TRUE; END_IF;

// Rung 170: G3_FAULT_RESET
// Reset fault dari panel
  LD %M351                (* SCADA_RESET_FAULT *)
  R %M4                   (* FAULT_G3 *)
  // as ST:
  //   IF SCADA_RESET_FAULT THEN FAULT_G3 := FALSE; END_IF;

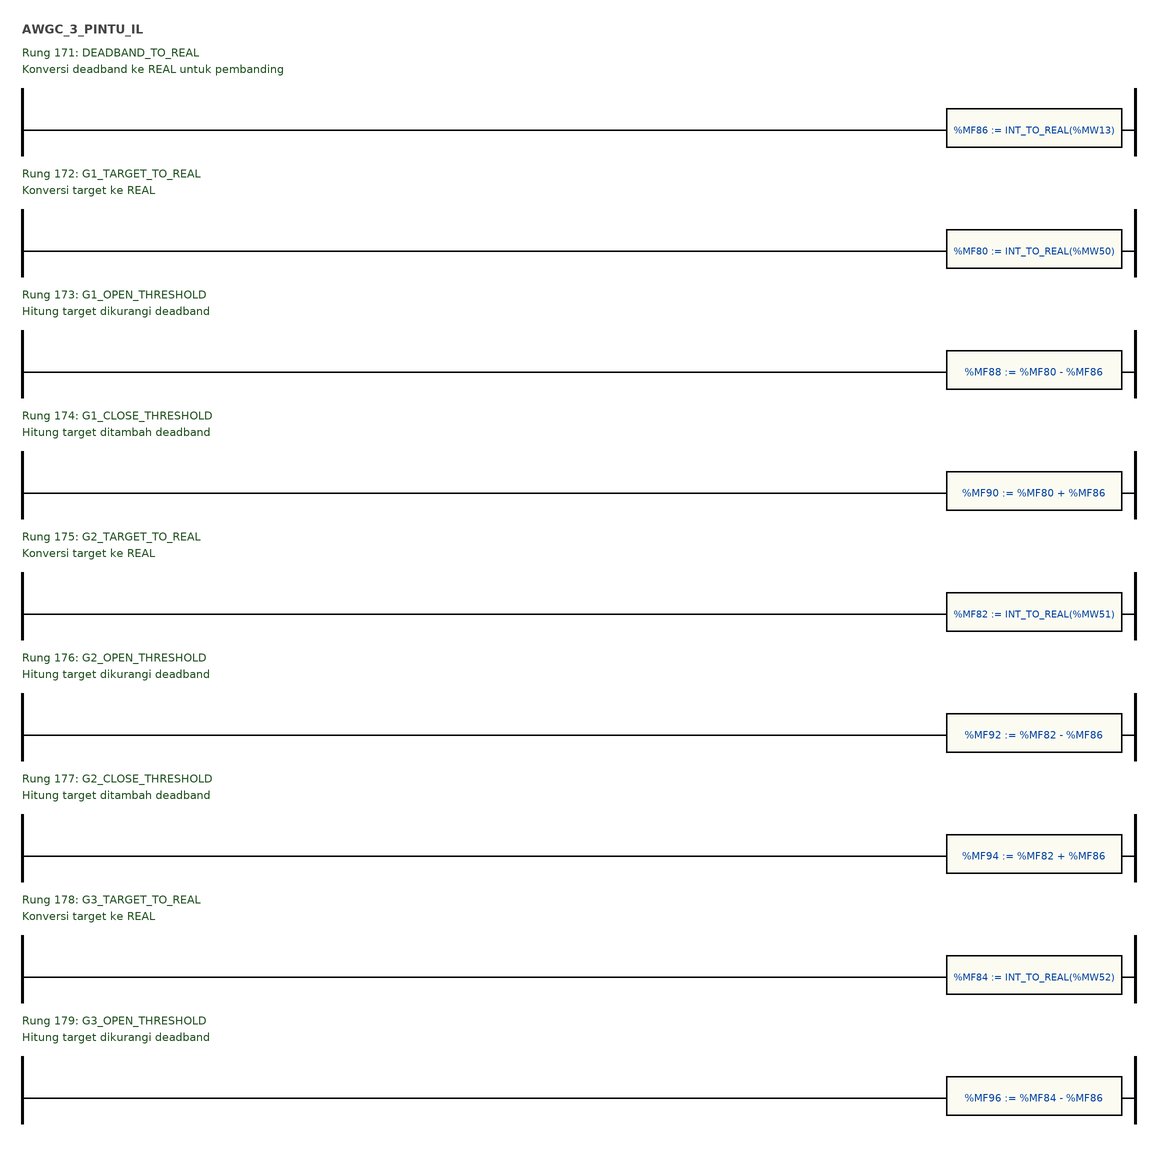

// Rung 171: DEADBAND_TO_REAL
// Konversi deadband ke REAL untuk pembanding
  LD 1
  [ %MF86 := INT_TO_REAL ( %MW13 ) ](* DEADBAND_REAL, DEADBAND_PCT *)
  // as ST:
  //   DEADBAND_REAL := INT_TO_REAL ( DEADBAND_PCT );

// Rung 172: G1_TARGET_TO_REAL
// Konversi target ke REAL
  LD 1
  [ %MF80 := INT_TO_REAL ( %MW50 ) ](* TARGET_G1_REAL, TARGET_PCT_G1 *)
  // as ST:
  //   TARGET_G1_REAL := INT_TO_REAL ( TARGET_PCT_G1 );

// Rung 173: G1_OPEN_THRESHOLD
// Hitung target dikurangi deadband
  LD 1
  [ %MF88 := %MF80 - %MF86 ](* OPEN_THRESHOLD_G1, TARGET_G1_REAL, DEADBAND_REAL *)
  // as ST:
  //   OPEN_THRESHOLD_G1 := TARGET_G1_REAL - DEADBAND_REAL;

// Rung 174: G1_CLOSE_THRESHOLD
// Hitung target ditambah deadband
  LD 1
  [ %MF90 := %MF80 + %MF86 ](* CLOSE_THRESHOLD_G1, TARGET_G1_REAL, DEADBAND_REAL *)
  // as ST:
  //   CLOSE_THRESHOLD_G1 := TARGET_G1_REAL + DEADBAND_REAL;

// Rung 175: G2_TARGET_TO_REAL
// Konversi target ke REAL
  LD 1
  [ %MF82 := INT_TO_REAL ( %MW51 ) ](* TARGET_G2_REAL, TARGET_PCT_G2 *)
  // as ST:
  //   TARGET_G2_REAL := INT_TO_REAL ( TARGET_PCT_G2 );

// Rung 176: G2_OPEN_THRESHOLD
// Hitung target dikurangi deadband
  LD 1
  [ %MF92 := %MF82 - %MF86 ](* OPEN_THRESHOLD_G2, TARGET_G2_REAL, DEADBAND_REAL *)
  // as ST:
  //   OPEN_THRESHOLD_G2 := TARGET_G2_REAL - DEADBAND_REAL;

// Rung 177: G2_CLOSE_THRESHOLD
// Hitung target ditambah deadband
  LD 1
  [ %MF94 := %MF82 + %MF86 ](* CLOSE_THRESHOLD_G2, TARGET_G2_REAL, DEADBAND_REAL *)
  // as ST:
  //   CLOSE_THRESHOLD_G2 := TARGET_G2_REAL + DEADBAND_REAL;

// Rung 178: G3_TARGET_TO_REAL
// Konversi target ke REAL
  LD 1
  [ %MF84 := INT_TO_REAL ( %MW52 ) ](* TARGET_G3_REAL, TARGET_PCT_G3 *)
  // as ST:
  //   TARGET_G3_REAL := INT_TO_REAL ( TARGET_PCT_G3 );

// Rung 179: G3_OPEN_THRESHOLD
// Hitung target dikurangi deadband
  LD 1
  [ %MF96 := %MF84 - %MF86 ](* OPEN_THRESHOLD_G3, TARGET_G3_REAL, DEADBAND_REAL *)
  // as ST:
  //   OPEN_THRESHOLD_G3 := TARGET_G3_REAL - DEADBAND_REAL;

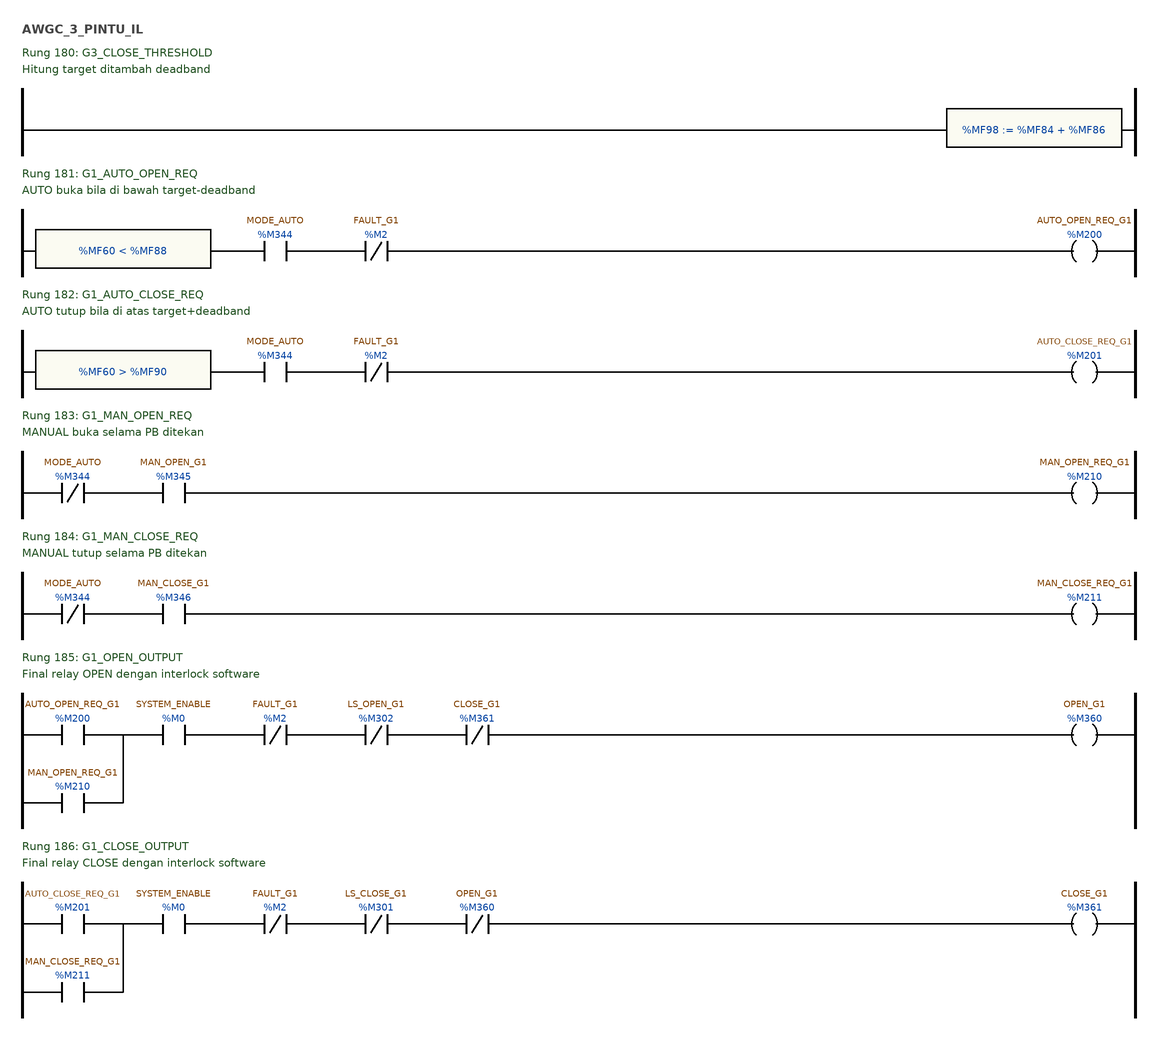

// Rung 180: G3_CLOSE_THRESHOLD
// Hitung target ditambah deadband
  LD 1
  [ %MF98 := %MF84 + %MF86 ](* CLOSE_THRESHOLD_G3, TARGET_G3_REAL, DEADBAND_REAL *)
  // as ST:
  //   CLOSE_THRESHOLD_G3 := TARGET_G3_REAL + DEADBAND_REAL;

// Rung 181: G1_AUTO_OPEN_REQ
// AUTO buka bila di bawah target-deadband
  LD [ %MF60 < %MF88 ]    (* POSITION_G1_PCT, OPEN_THRESHOLD_G1 *)
  AND %M344               (* SCADA_MODE_AUTO *)
  ANDN %M2                (* FAULT_G1 *)
  ST %M200                (* AUTO_OPEN_REQ_G1 *)
  // as ST:
  //   AUTO_OPEN_REQ_G1 := POSITION_G1_PCT < OPEN_THRESHOLD_G1 AND SCADA_MODE_AUTO AND NOT FAULT_G1;

// Rung 182: G1_AUTO_CLOSE_REQ
// AUTO tutup bila di atas target+deadband
  LD [ %MF60 > %MF90 ]    (* POSITION_G1_PCT, CLOSE_THRESHOLD_G1 *)
  AND %M344               (* SCADA_MODE_AUTO *)
  ANDN %M2                (* FAULT_G1 *)
  ST %M201                (* AUTO_CLOSE_REQ_G1 *)
  // as ST:
  //   AUTO_CLOSE_REQ_G1 := POSITION_G1_PCT > CLOSE_THRESHOLD_G1 AND SCADA_MODE_AUTO AND NOT FAULT_G1;

// Rung 183: G1_MAN_OPEN_REQ
// MANUAL buka selama PB ditekan
  LDN %M344               (* SCADA_MODE_AUTO *)
  AND %M345               (* SIM_I1_25 *)
  ST %M210                (* MAN_OPEN_REQ_G1 *)
  // as ST:
  //   MAN_OPEN_REQ_G1 := NOT SCADA_MODE_AUTO AND SIM_I1_25;

// Rung 184: G1_MAN_CLOSE_REQ
// MANUAL tutup selama PB ditekan
  LDN %M344               (* SCADA_MODE_AUTO *)
  AND %M346               (* SIM_I1_26 *)
  ST %M211                (* MAN_CLOSE_REQ_G1 *)
  // as ST:
  //   MAN_CLOSE_REQ_G1 := NOT SCADA_MODE_AUTO AND SIM_I1_26;

// Rung 185: G1_OPEN_OUTPUT
// Final relay OPEN dengan interlock software
  LD %M200                (* AUTO_OPEN_REQ_G1 *)
  OR %M210                (* MAN_OPEN_REQ_G1 *)
  AND %M0                 (* SYSTEM_ENABLE *)
  ANDN %M2                (* FAULT_G1 *)
  ANDN %M302              (* SCADA_LS_OPEN_G1 *)
  ANDN %M361              (* SIM_Q0_1 *)
  ST %M360                (* SIM_Q0_0 *)
  // as ST:
  //   SIM_Q0_0 := (AUTO_OPEN_REQ_G1 OR MAN_OPEN_REQ_G1) AND SYSTEM_ENABLE AND NOT FAULT_G1 AND NOT SCADA_LS_OPEN_G1 AND NOT SIM_Q0_1;

// Rung 186: G1_CLOSE_OUTPUT
// Final relay CLOSE dengan interlock software
  LD %M201                (* AUTO_CLOSE_REQ_G1 *)
  OR %M211                (* MAN_CLOSE_REQ_G1 *)
  AND %M0                 (* SYSTEM_ENABLE *)
  ANDN %M2                (* FAULT_G1 *)
  ANDN %M301              (* SCADA_LS_CLOSE_G1 *)
  ANDN %M360              (* SIM_Q0_0 *)
  ST %M361                (* SIM_Q0_1 *)
  // as ST:
  //   SIM_Q0_1 := (AUTO_CLOSE_REQ_G1 OR MAN_CLOSE_REQ_G1) AND SYSTEM_ENABLE AND NOT FAULT_G1 AND NOT SCADA_LS_CLOSE_G1 AND NOT SIM_Q0_0;

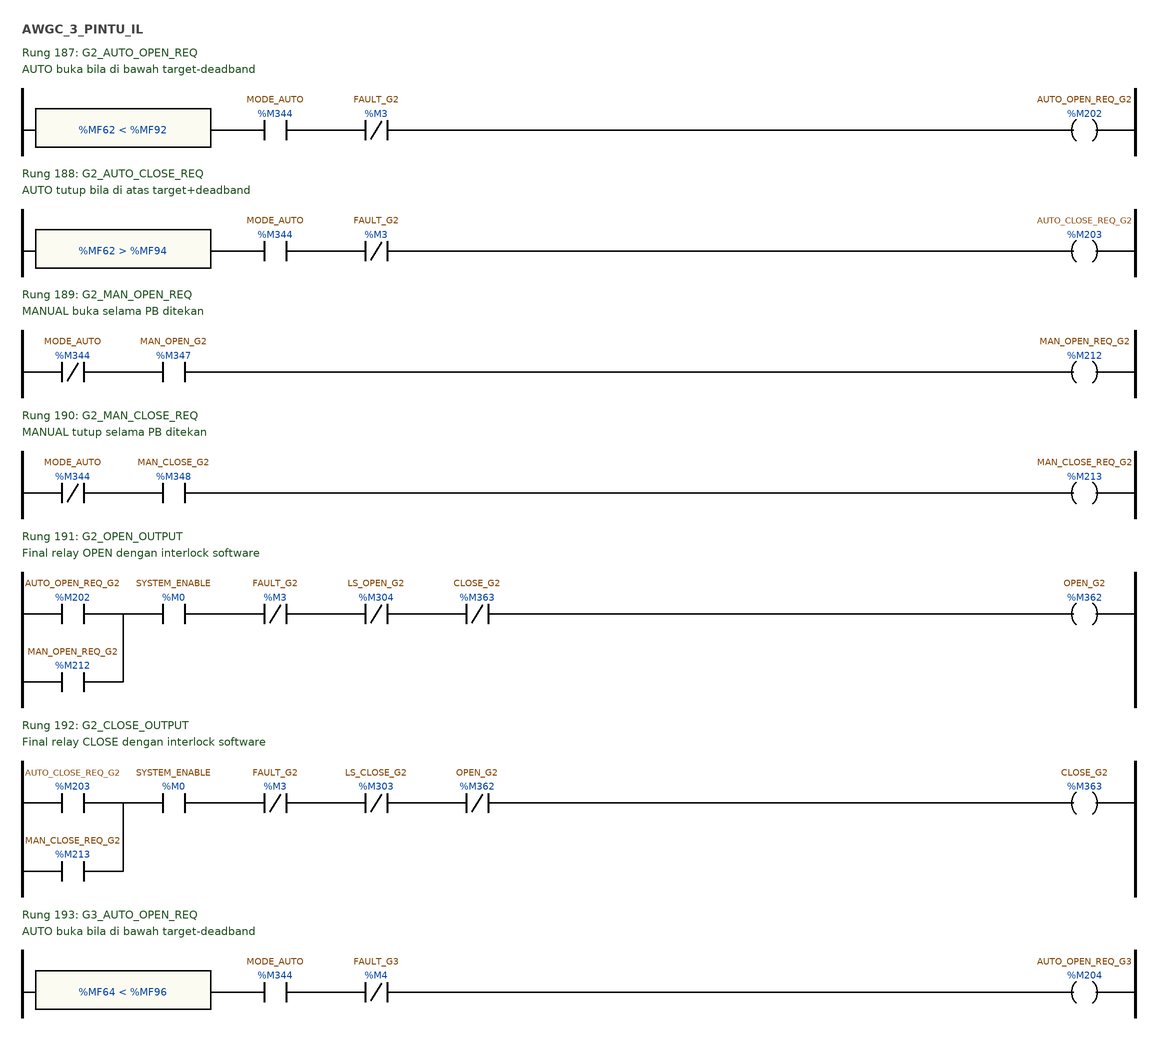

// Rung 187: G2_AUTO_OPEN_REQ
// AUTO buka bila di bawah target-deadband
  LD [ %MF62 < %MF92 ]    (* POSITION_G2_PCT, OPEN_THRESHOLD_G2 *)
  AND %M344               (* SCADA_MODE_AUTO *)
  ANDN %M3                (* FAULT_G2 *)
  ST %M202                (* AUTO_OPEN_REQ_G2 *)
  // as ST:
  //   AUTO_OPEN_REQ_G2 := POSITION_G2_PCT < OPEN_THRESHOLD_G2 AND SCADA_MODE_AUTO AND NOT FAULT_G2;

// Rung 188: G2_AUTO_CLOSE_REQ
// AUTO tutup bila di atas target+deadband
  LD [ %MF62 > %MF94 ]    (* POSITION_G2_PCT, CLOSE_THRESHOLD_G2 *)
  AND %M344               (* SCADA_MODE_AUTO *)
  ANDN %M3                (* FAULT_G2 *)
  ST %M203                (* AUTO_CLOSE_REQ_G2 *)
  // as ST:
  //   AUTO_CLOSE_REQ_G2 := POSITION_G2_PCT > CLOSE_THRESHOLD_G2 AND SCADA_MODE_AUTO AND NOT FAULT_G2;

// Rung 189: G2_MAN_OPEN_REQ
// MANUAL buka selama PB ditekan
  LDN %M344               (* SCADA_MODE_AUTO *)
  AND %M347               (* SIM_I1_27 *)
  ST %M212                (* MAN_OPEN_REQ_G2 *)
  // as ST:
  //   MAN_OPEN_REQ_G2 := NOT SCADA_MODE_AUTO AND SIM_I1_27;

// Rung 190: G2_MAN_CLOSE_REQ
// MANUAL tutup selama PB ditekan
  LDN %M344               (* SCADA_MODE_AUTO *)
  AND %M348               (* SIM_I1_28 *)
  ST %M213                (* MAN_CLOSE_REQ_G2 *)
  // as ST:
  //   MAN_CLOSE_REQ_G2 := NOT SCADA_MODE_AUTO AND SIM_I1_28;

// Rung 191: G2_OPEN_OUTPUT
// Final relay OPEN dengan interlock software
  LD %M202                (* AUTO_OPEN_REQ_G2 *)
  OR %M212                (* MAN_OPEN_REQ_G2 *)
  AND %M0                 (* SYSTEM_ENABLE *)
  ANDN %M3                (* FAULT_G2 *)
  ANDN %M304              (* SCADA_LS_OPEN_G2 *)
  ANDN %M363              (* SIM_Q0_3 *)
  ST %M362                (* SIM_Q0_2 *)
  // as ST:
  //   SIM_Q0_2 := (AUTO_OPEN_REQ_G2 OR MAN_OPEN_REQ_G2) AND SYSTEM_ENABLE AND NOT FAULT_G2 AND NOT SCADA_LS_OPEN_G2 AND NOT SIM_Q0_3;

// Rung 192: G2_CLOSE_OUTPUT
// Final relay CLOSE dengan interlock software
  LD %M203                (* AUTO_CLOSE_REQ_G2 *)
  OR %M213                (* MAN_CLOSE_REQ_G2 *)
  AND %M0                 (* SYSTEM_ENABLE *)
  ANDN %M3                (* FAULT_G2 *)
  ANDN %M303              (* SCADA_LS_CLOSE_G2 *)
  ANDN %M362              (* SIM_Q0_2 *)
  ST %M363                (* SIM_Q0_3 *)
  // as ST:
  //   SIM_Q0_3 := (AUTO_CLOSE_REQ_G2 OR MAN_CLOSE_REQ_G2) AND SYSTEM_ENABLE AND NOT FAULT_G2 AND NOT SCADA_LS_CLOSE_G2 AND NOT SIM_Q0_2;

// Rung 193: G3_AUTO_OPEN_REQ
// AUTO buka bila di bawah target-deadband
  LD [ %MF64 < %MF96 ]    (* POSITION_G3_PCT, OPEN_THRESHOLD_G3 *)
  AND %M344               (* SCADA_MODE_AUTO *)
  ANDN %M4                (* FAULT_G3 *)
  ST %M204                (* AUTO_OPEN_REQ_G3 *)
  // as ST:
  //   AUTO_OPEN_REQ_G3 := POSITION_G3_PCT < OPEN_THRESHOLD_G3 AND SCADA_MODE_AUTO AND NOT FAULT_G3;

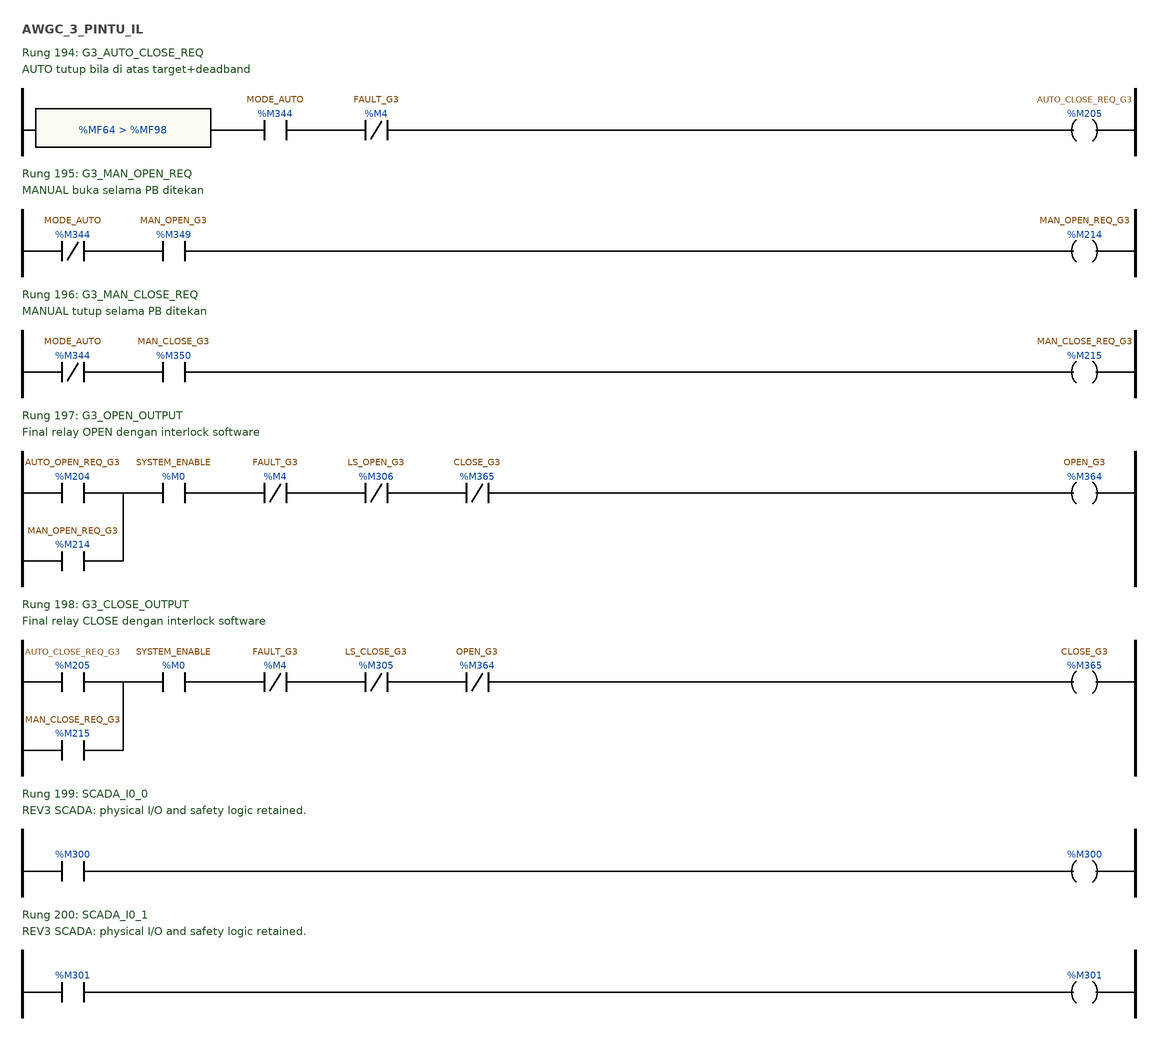

// Rung 194: G3_AUTO_CLOSE_REQ
// AUTO tutup bila di atas target+deadband
  LD [ %MF64 > %MF98 ]    (* POSITION_G3_PCT, CLOSE_THRESHOLD_G3 *)
  AND %M344               (* SCADA_MODE_AUTO *)
  ANDN %M4                (* FAULT_G3 *)
  ST %M205                (* AUTO_CLOSE_REQ_G3 *)
  // as ST:
  //   AUTO_CLOSE_REQ_G3 := POSITION_G3_PCT > CLOSE_THRESHOLD_G3 AND SCADA_MODE_AUTO AND NOT FAULT_G3;

// Rung 195: G3_MAN_OPEN_REQ
// MANUAL buka selama PB ditekan
  LDN %M344               (* SCADA_MODE_AUTO *)
  AND %M349               (* SIM_I1_29 *)
  ST %M214                (* MAN_OPEN_REQ_G3 *)
  // as ST:
  //   MAN_OPEN_REQ_G3 := NOT SCADA_MODE_AUTO AND SIM_I1_29;

// Rung 196: G3_MAN_CLOSE_REQ
// MANUAL tutup selama PB ditekan
  LDN %M344               (* SCADA_MODE_AUTO *)
  AND %M350               (* SIM_I1_30 *)
  ST %M215                (* MAN_CLOSE_REQ_G3 *)
  // as ST:
  //   MAN_CLOSE_REQ_G3 := NOT SCADA_MODE_AUTO AND SIM_I1_30;

// Rung 197: G3_OPEN_OUTPUT
// Final relay OPEN dengan interlock software
  LD %M204                (* AUTO_OPEN_REQ_G3 *)
  OR %M214                (* MAN_OPEN_REQ_G3 *)
  AND %M0                 (* SYSTEM_ENABLE *)
  ANDN %M4                (* FAULT_G3 *)
  ANDN %M306              (* SCADA_LS_OPEN_G3 *)
  ANDN %M365              (* SIM_Q0_5 *)
  ST %M364                (* SIM_Q0_4 *)
  // as ST:
  //   SIM_Q0_4 := (AUTO_OPEN_REQ_G3 OR MAN_OPEN_REQ_G3) AND SYSTEM_ENABLE AND NOT FAULT_G3 AND NOT SCADA_LS_OPEN_G3 AND NOT SIM_Q0_5;

// Rung 198: G3_CLOSE_OUTPUT
// Final relay CLOSE dengan interlock software
  LD %M205                (* AUTO_CLOSE_REQ_G3 *)
  OR %M215                (* MAN_CLOSE_REQ_G3 *)
  AND %M0                 (* SYSTEM_ENABLE *)
  ANDN %M4                (* FAULT_G3 *)
  ANDN %M305              (* SCADA_LS_CLOSE_G3 *)
  ANDN %M364              (* SIM_Q0_4 *)
  ST %M365                (* SIM_Q0_5 *)
  // as ST:
  //   SIM_Q0_5 := (AUTO_CLOSE_REQ_G3 OR MAN_CLOSE_REQ_G3) AND SYSTEM_ENABLE AND NOT FAULT_G3 AND NOT SCADA_LS_CLOSE_G3 AND NOT SIM_Q0_4;

// Rung 199: SCADA_I0_0
// REV3 SCADA: physical I/O and safety logic retained.
  LD %M300                (* SCADA_SAFETY_OK *)
  ST %M300                (* SCADA_SAFETY_OK *)
  // as ST:
  //   SCADA_SAFETY_OK := SCADA_SAFETY_OK;

// Rung 200: SCADA_I0_1
// REV3 SCADA: physical I/O and safety logic retained.
  LD %M301                (* SCADA_LS_CLOSE_G1 *)
  ST %M301                (* SCADA_LS_CLOSE_G1 *)
  // as ST:
  //   SCADA_LS_CLOSE_G1 := SCADA_LS_CLOSE_G1;

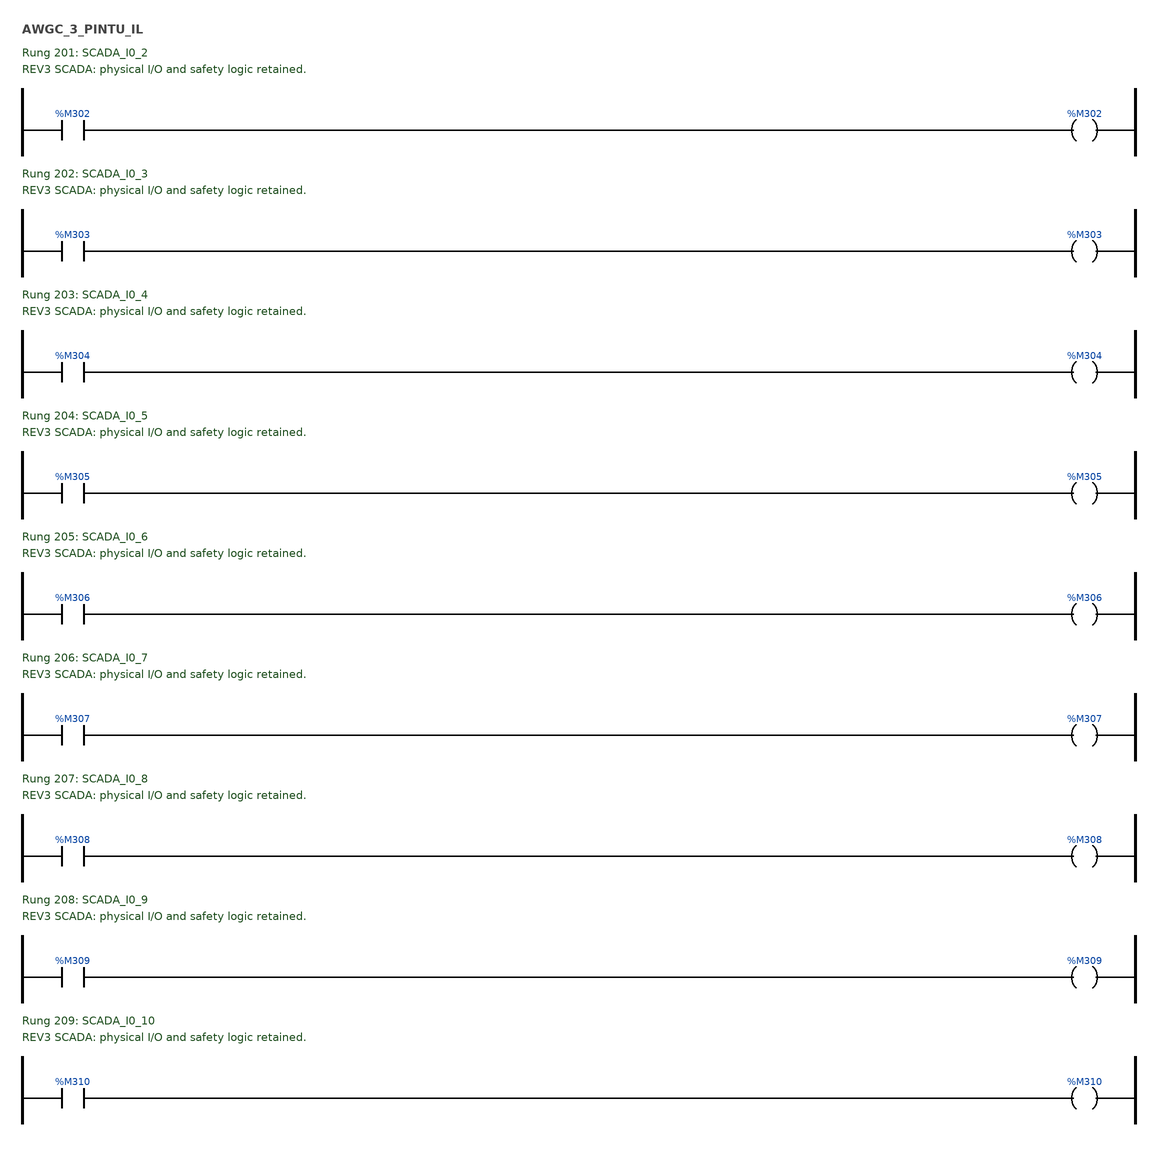

// Rung 201: SCADA_I0_2
// REV3 SCADA: physical I/O and safety logic retained.
  LD %M302                (* SCADA_LS_OPEN_G1 *)
  ST %M302                (* SCADA_LS_OPEN_G1 *)
  // as ST:
  //   SCADA_LS_OPEN_G1 := SCADA_LS_OPEN_G1;

// Rung 202: SCADA_I0_3
// REV3 SCADA: physical I/O and safety logic retained.
  LD %M303                (* SCADA_LS_CLOSE_G2 *)
  ST %M303                (* SCADA_LS_CLOSE_G2 *)
  // as ST:
  //   SCADA_LS_CLOSE_G2 := SCADA_LS_CLOSE_G2;

// Rung 203: SCADA_I0_4
// REV3 SCADA: physical I/O and safety logic retained.
  LD %M304                (* SCADA_LS_OPEN_G2 *)
  ST %M304                (* SCADA_LS_OPEN_G2 *)
  // as ST:
  //   SCADA_LS_OPEN_G2 := SCADA_LS_OPEN_G2;

// Rung 204: SCADA_I0_5
// REV3 SCADA: physical I/O and safety logic retained.
  LD %M305                (* SCADA_LS_CLOSE_G3 *)
  ST %M305                (* SCADA_LS_CLOSE_G3 *)
  // as ST:
  //   SCADA_LS_CLOSE_G3 := SCADA_LS_CLOSE_G3;

// Rung 205: SCADA_I0_6
// REV3 SCADA: physical I/O and safety logic retained.
  LD %M306                (* SCADA_LS_OPEN_G3 *)
  ST %M306                (* SCADA_LS_OPEN_G3 *)
  // as ST:
  //   SCADA_LS_OPEN_G3 := SCADA_LS_OPEN_G3;

// Rung 206: SCADA_I0_7
// REV3 SCADA: physical I/O and safety logic retained.
  LD %M307                (* SCADA_OL_G1_OK *)
  ST %M307                (* SCADA_OL_G1_OK *)
  // as ST:
  //   SCADA_OL_G1_OK := SCADA_OL_G1_OK;

// Rung 207: SCADA_I0_8
// REV3 SCADA: physical I/O and safety logic retained.
  LD %M308                (* SCADA_OL_G2_OK *)
  ST %M308                (* SCADA_OL_G2_OK *)
  // as ST:
  //   SCADA_OL_G2_OK := SCADA_OL_G2_OK;

// Rung 208: SCADA_I0_9
// REV3 SCADA: physical I/O and safety logic retained.
  LD %M309                (* SCADA_OL_G3_OK *)
  ST %M309                (* SCADA_OL_G3_OK *)
  // as ST:
  //   SCADA_OL_G3_OK := SCADA_OL_G3_OK;

// Rung 209: SCADA_I0_10
// REV3 SCADA: physical I/O and safety logic retained.
  LD %M310                (* SIM_I0_10 *)
  ST %M310                (* SIM_I0_10 *)
  // as ST:
  //   SIM_I0_10 := SIM_I0_10;

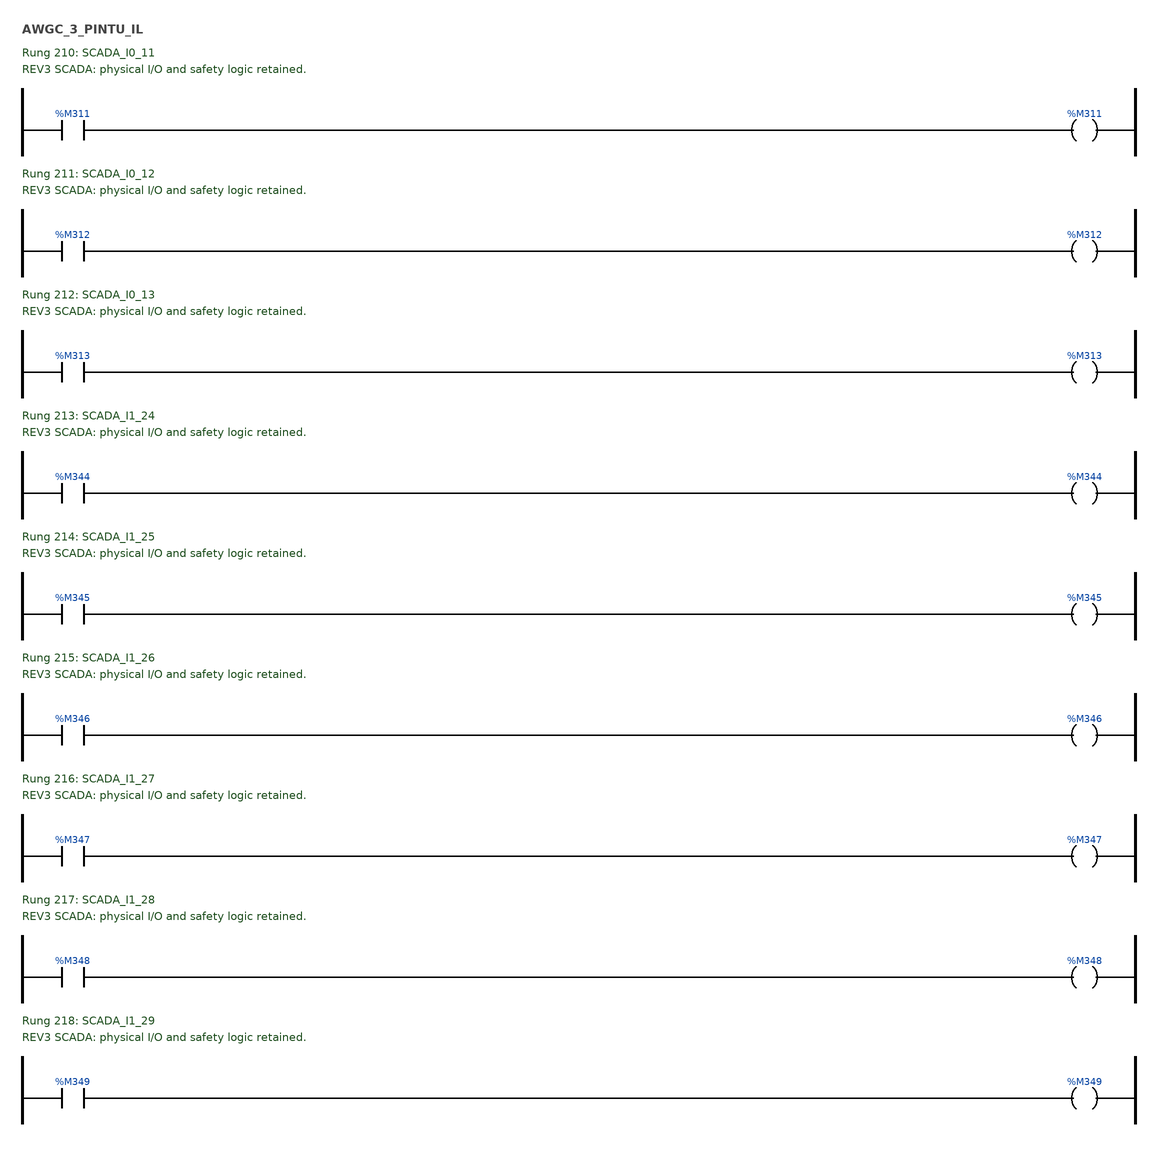

// Rung 210: SCADA_I0_11
// REV3 SCADA: physical I/O and safety logic retained.
  LD %M311                (* SIM_I0_11 *)
  ST %M311                (* SIM_I0_11 *)
  // as ST:
  //   SIM_I0_11 := SIM_I0_11;

// Rung 211: SCADA_I0_12
// REV3 SCADA: physical I/O and safety logic retained.
  LD %M312                (* SIM_I0_12 *)
  ST %M312                (* SIM_I0_12 *)
  // as ST:
  //   SIM_I0_12 := SIM_I0_12;

// Rung 212: SCADA_I0_13
// REV3 SCADA: physical I/O and safety logic retained.
  LD %M313                (* SIM_I0_13 *)
  ST %M313                (* SIM_I0_13 *)
  // as ST:
  //   SIM_I0_13 := SIM_I0_13;

// Rung 213: SCADA_I1_24
// REV3 SCADA: physical I/O and safety logic retained.
  LD %M344                (* SCADA_MODE_AUTO *)
  ST %M344                (* SCADA_MODE_AUTO *)
  // as ST:
  //   SCADA_MODE_AUTO := SCADA_MODE_AUTO;

// Rung 214: SCADA_I1_25
// REV3 SCADA: physical I/O and safety logic retained.
  LD %M345                (* SIM_I1_25 *)
  ST %M345                (* SIM_I1_25 *)
  // as ST:
  //   SIM_I1_25 := SIM_I1_25;

// Rung 215: SCADA_I1_26
// REV3 SCADA: physical I/O and safety logic retained.
  LD %M346                (* SIM_I1_26 *)
  ST %M346                (* SIM_I1_26 *)
  // as ST:
  //   SIM_I1_26 := SIM_I1_26;

// Rung 216: SCADA_I1_27
// REV3 SCADA: physical I/O and safety logic retained.
  LD %M347                (* SIM_I1_27 *)
  ST %M347                (* SIM_I1_27 *)
  // as ST:
  //   SIM_I1_27 := SIM_I1_27;

// Rung 217: SCADA_I1_28
// REV3 SCADA: physical I/O and safety logic retained.
  LD %M348                (* SIM_I1_28 *)
  ST %M348                (* SIM_I1_28 *)
  // as ST:
  //   SIM_I1_28 := SIM_I1_28;

// Rung 218: SCADA_I1_29
// REV3 SCADA: physical I/O and safety logic retained.
  LD %M349                (* SIM_I1_29 *)
  ST %M349                (* SIM_I1_29 *)
  // as ST:
  //   SIM_I1_29 := SIM_I1_29;

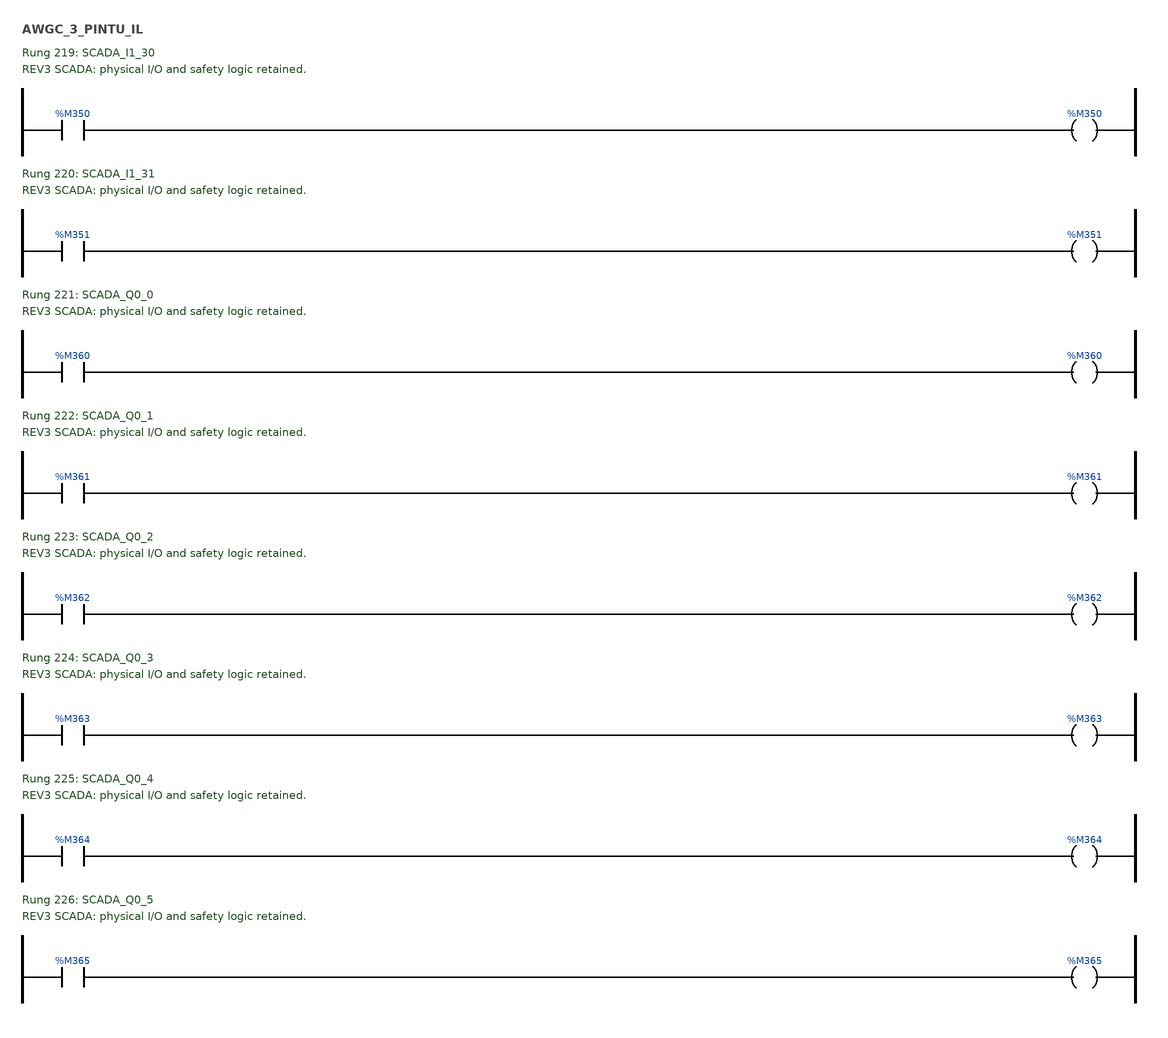

// Rung 219: SCADA_I1_30
// REV3 SCADA: physical I/O and safety logic retained.
  LD %M350                (* SIM_I1_30 *)
  ST %M350                (* SIM_I1_30 *)
  // as ST:
  //   SIM_I1_30 := SIM_I1_30;

// Rung 220: SCADA_I1_31
// REV3 SCADA: physical I/O and safety logic retained.
  LD %M351                (* SCADA_RESET_FAULT *)
  ST %M351                (* SCADA_RESET_FAULT *)
  // as ST:
  //   SCADA_RESET_FAULT := SCADA_RESET_FAULT;

// Rung 221: SCADA_Q0_0
// REV3 SCADA: physical I/O and safety logic retained.
  LD %M360                (* SIM_Q0_0 *)
  ST %M360                (* SIM_Q0_0 *)
  // as ST:
  //   SIM_Q0_0 := SIM_Q0_0;

// Rung 222: SCADA_Q0_1
// REV3 SCADA: physical I/O and safety logic retained.
  LD %M361                (* SIM_Q0_1 *)
  ST %M361                (* SIM_Q0_1 *)
  // as ST:
  //   SIM_Q0_1 := SIM_Q0_1;

// Rung 223: SCADA_Q0_2
// REV3 SCADA: physical I/O and safety logic retained.
  LD %M362                (* SIM_Q0_2 *)
  ST %M362                (* SIM_Q0_2 *)
  // as ST:
  //   SIM_Q0_2 := SIM_Q0_2;

// Rung 224: SCADA_Q0_3
// REV3 SCADA: physical I/O and safety logic retained.
  LD %M363                (* SIM_Q0_3 *)
  ST %M363                (* SIM_Q0_3 *)
  // as ST:
  //   SIM_Q0_3 := SIM_Q0_3;

// Rung 225: SCADA_Q0_4
// REV3 SCADA: physical I/O and safety logic retained.
  LD %M364                (* SIM_Q0_4 *)
  ST %M364                (* SIM_Q0_4 *)
  // as ST:
  //   SIM_Q0_4 := SIM_Q0_4;

// Rung 226: SCADA_Q0_5
// REV3 SCADA: physical I/O and safety logic retained.
  LD %M365                (* SIM_Q0_5 *)
  ST %M365                (* SIM_Q0_5 *)
  // as ST:
  //   SIM_Q0_5 := SIM_Q0_5;

// Rung 227: PHYSICAL_OUTPUT_0_LOCKED_OFF
// SIMULATOR ONLY. Physical outputs forced OFF. Do not use for plant operation.
  LD 0
  ST %Q0.0                (* OPEN_G1 *)
  // as ST:
  //   OPEN_G1 := FALSE;

// Rung 228: PHYSICAL_OUTPUT_1_LOCKED_OFF
// SIMULATOR ONLY. Physical outputs forced OFF. Do not use for plant operation.
  LD 0
  ST %Q0.1                (* CLOSE_G1 *)
  // as ST:
  //   CLOSE_G1 := FALSE;

// Rung 229: PHYSICAL_OUTPUT_2_LOCKED_OFF
// SIMULATOR ONLY. Physical outputs forced OFF. Do not use for plant operation.
  LD 0
  ST %Q0.2                (* OPEN_G2 *)
  // as ST:
  //   OPEN_G2 := FALSE;

// Rung 230: PHYSICAL_OUTPUT_3_LOCKED_OFF
// SIMULATOR ONLY. Physical outputs forced OFF. Do not use for plant operation.
  LD 0
  ST %Q0.3                (* CLOSE_G2 *)
  // as ST:
  //   CLOSE_G2 := FALSE;

// Rung 231: PHYSICAL_OUTPUT_4_LOCKED_OFF
// SIMULATOR ONLY. Physical outputs forced OFF. Do not use for plant operation.
  LD 0
  ST %Q0.4                (* OPEN_G3 *)
  // as ST:
  //   OPEN_G3 := FALSE;

// Rung 232: PHYSICAL_OUTPUT_5_LOCKED_OFF
// SIMULATOR ONLY. Physical outputs forced OFF. Do not use for plant operation.
  LD 0
  ST %Q0.5                (* CLOSE_G3 *)
  // as ST:
  //   CLOSE_G3 := FALSE;

// Rung 233: PHYSICAL_OUTPUT_6_LOCKED_OFF
// SIMULATOR ONLY. Physical outputs forced OFF. Do not use for plant operation.
  LD 0
  ST %Q0.6
  // as ST:
  //   %Q0.6 := FALSE;

// Rung 234: PHYSICAL_OUTPUT_7_LOCKED_OFF
// SIMULATOR ONLY. Physical outputs forced OFF. Do not use for plant operation.
  LD 0
  ST %Q0.7
  // as ST:
  //   %Q0.7 := FALSE;

// Rung 235: PHYSICAL_OUTPUT_8_LOCKED_OFF
// SIMULATOR ONLY. Physical outputs forced OFF. Do not use for plant operation.
  LD 0
  ST %Q0.8
  // as ST:
  //   %Q0.8 := FALSE;

// Rung 236: PHYSICAL_OUTPUT_9_LOCKED_OFF
// SIMULATOR ONLY. Physical outputs forced OFF. Do not use for plant operation.
  LD 0
  ST %Q0.9
  // as ST:
  //   %Q0.9 := FALSE;
